# B&R Automation Studio project x20ost (part 8)

#### bnrtcpserver.c
```c
/********************************************************************
 * COPYRIGHT -- Kontora
 ********************************************************************
 * Program: bnrmain
 * File: bnrlsens.c
 * Author: Abramenya
 * Created: January 19, 2009
 *******************************************************************/

#include "bnrtcpserver.h"
#ifdef _DEFAULT_INCLUDES
 #include <AsDefault.h>
#endif
#ifdef WIN32
DWORD dwThreadId;
//void TcpOpen(TcpOpen_typ *pServer){pServer->status=0;}
SOCKET sClient;
DWORD WINAPI GetArm(PVOID pVoid);
void TcpClose(TcpClose_typ *pCL){};
void TcpServer(TcpServer_typ *pServer){pServer->identclnt=pServer->ident;pServer->status=0;}
void TcpOpen(TcpOpen_typ *pServer)
{
	BOOL    bInterface = FALSE;
    WSADATA wsd;
	int iAddrSize;
	struct sockaddr_in local,client;
	struct sockaddr_in server;
    struct hostent *host = NULL;
	pServer->status = 1;
	if (WSAStartup(MAKEWORD(2,2), &wsd) != 0)
    {
        printf("Failed to load Winsock!\n");
        return ;
    }
	pServer->sListen = socket(AF_INET, SOCK_STREAM, IPPROTO_TCP);
    if (pServer->sListen == SOCKET_ERROR)
    {
        printf("socket() failed: %d\n", WSAGetLastError());
        return ;
    }
    if (bInterface)
    {
        //local.sin_addr.s_addr = inet_addr(pServer->pIfAddr);
		local.sin_addr.s_addr = inet_addr("0.0.0.0");
        if (local.sin_addr.s_addr == INADDR_NONE)
		{
			printf("socket() failed: %s\n", pServer->pIfAddr);
			return;
		}
    }
    else
		local.sin_addr.s_addr = htonl(INADDR_ANY);
	local.sin_family = AF_INET;
	local.sin_port = htons((u_short)pServer->port);
    if (bind(pServer->sListen, (struct sockaddr *)&local,sizeof(local)) == SOCKET_ERROR)
    {
        printf("bind() failed: %d\n", WSAGetLastError());
        return ;
    }
    listen(pServer->sListen, 8);
    iAddrSize = sizeof(client);
    //pServer->sClient = accept(pServer->sListen, (struct sockaddr *)&client,&iAddrSize);
	pServer->sClient = accept(pServer->sListen, (struct sockaddr *)&client,&iAddrSize);
    if (pServer->sClient == INVALID_SOCKET)
    {
		printf("accept() failed: %d\n", WSAGetLastError());
		return ;
    }
	sClient = pServer->sClient;
	pServer->ident = &pServer->sClient;
	Info("\n(__)CTCPS::>Connect");
	pServer->status = 0;
}
//void TcpSend(TcpSend_typ *pCL){};
void TcpSend(TcpSend_typ *pSend)
{
	int ret;
	ret = send(sClient, (char*)pSend->pData, pSend->datalen, 0);
	//Info("\n(__)ARM_0:%M",pSend->buffer);
	if (ret == 0)
	{
		//printf("Send Not Poss \n");
		//Sleep(500);
		pSend->status = 1;
		return;
	}
	else if (ret == SOCKET_ERROR)
	{
		//printf("send() failed: %d\n",WSAGetLastError());
		//Sleep(500);
		pSend->status = 1;
		return;
	}
	//Sleep(50);
	pSend->status = 0;

}
void TcpRecv(TcpRecv_typ *pRecv)
{
	int ret;
	//printf("RCV\n");
	ret = recv(sClient,(char*)pRecv->pData,pRecv->datamax , 0);
	if (ret == 0)
	{
		//Sleep(500);
		printf("recv() failed 0: %d\n", WSAGetLastError());
		pRecv->status = 1;
		return;
	}
	else if (ret == SOCKET_ERROR)
	{
		printf("recv() failed: %d\n", WSAGetLastError());
        //Sleep(500);
		pRecv->status = 1;
		return;
	}
	//printf("Reccive OK! \n");
	pRecv->recvlen = ret;
	pRecv->status = 0;
}
#endif

//_GLOBAL INT iCreate1;
_GLOBAL UINT iCreateTcp1;
void CTcpServer_Init(This,SARMINTERFACE *pArm)
{
    DECLARE_MULTI_OPEN(CTcpServer,CCyclicSystem)
	FDEFINE(DEV_TCPRM_BOX_ID,1024);
	FDEFINE(DEV_TCPBF_BOX_ID,1024);
	pB->SetBoxID(pB,DEV_TCPRM_BOX_ID);
	InitObject(CMTimer,&pT->m_nConnTMR);
	pT->m_nConnTMR.SetTimer(&pT->m_nConnTMR,DIR_TCPTOTCP,DIR_TCPTOTCP,EV_TMR_SRR_REQ,0,0,DEV_TCPRM_BOX_ID);
	pT->m_pArm = pArm;
	pT->m_dwAPortNumber = pArm->dwpPortNumber[0];
	pT->m_dwBPortNumber = pArm->dwpPortNumber[1];
	strcpy(pT->m_stTcpAddr,pArm->chTcpAddr);
	#ifdef DEB_CTcpServer
	Info("\n\r(__)CTcpS::>Create Tcp.PA: %d.PB: %d. Addr[%s]",&pT->m_dwAPortNumber,&pT->m_dwBPortNumber,pT->m_stTcpAddr);
    #endif
	memset(&pT->m_npListen,0,sizeof(TcpOpen_typ));
	memset(&pT->m_npServer,0,sizeof(TcpServer_typ));
	memset(&pT->m_npSend,0,sizeof(TcpSend_typ));
	pT->m_npListen.enable  = TRUE;
	pT->m_npListen.port    = pT->m_dwAPortNumber;
	pT->m_npListen.pIfAddr = 0;
	pT->m_npListen.status  = 1;
	pT->m_npListen.options = 0;

	pT->m_blSState = TRUE;
	pT->m_blRState = TRUE;
	pT->m_bSrvState = DRV_ST_DISC;

	pT->m_nConnTMR.OnTimer(&pT->m_nConnTMR,100);
    #ifdef WIN32
	CreateThread(NULL,0,GetArm ,pT,0,&dwThreadId);
	#endif
}
_GLOBAL TcpServer_typ sServer;
_GLOBAL TcpRecv_typ sRecc;
BOOL CTcpServer_Open(This)
{
	DECLARE_MULTI_OPEN(CTcpServer,CCyclicSystem)

	if(pT->m_bSrvState==DRV_ST_DISC)
	{
	 if (pT->m_byConnReq++%2==0)
	 {
	  pT->CloseRecc(pT);
	  pT->CloseSend(pT);
	  pT->CloseOpen(pT);
	 }
	 pT->Listen(pT);
	}

	if(pT->m_bSrvState==DRV_ST_OPEN)
	{
	 pT->m_npServer.enable  = 1;
	 pT->m_npServer.ident   = pT->m_npListen.ident;
	 pT->m_npServer.backlog = 1;
	 pT->m_npServer.pIpAddr = pT->m_stTcpAddr;
     TcpServer(&pT->m_npServer);
	 memcpy(&sServer,&pT->m_npServer,sizeof(TcpServer_typ));
     if(pT->m_npServer.status==0)
	 {

	  //if(pT->m_bSrvState==DRV_ST_OPEN)
      pT->m_npRecc.enable   = 1;
      pT->m_npRecc.ident    = pT->m_npServer.identclnt;
	  pT->m_npRecc.datamax  = sizeof(SMESSAGE)-10;
	  pT->m_npRecc.flags     = 0;

	  pT->m_npSend.enable   = 1;
	  pT->m_npSend.ident    = pT->m_npServer.identclnt;
	  pT->m_npSend.datalen  = sizeof(SMESSAGE);
	  pT->m_npSend.flags    = 0;
	  pT->m_bSrvState = DRV_ST_CONN;
	  pT->m_blSState = TRUE;
	  //pT->Connect(pT);
	  pT->SendSMessage(pT,DEV_KPMDL_BOX_ID,DIR_PHTOKP,PH_CALL_REQ);
  	  return TRUE;
	 }
	}
    return TRUE;
}
_GLOBAL TcpOpen_typ sOpen;
_GLOBAL INT iListen;
BOOL CTcpServer_Listen(This)
{
    DECLARE_MULTI_OPEN(CTcpServer,CCyclicSystem)
	iListen++;
	pT->m_npListen.enable  = TRUE;
	pT->m_npListen.port    = pT->m_dwAPortNumber;
	pT->m_npListen.pIfAddr = 0;
	pT->m_npListen.status  = 1;
	pT->m_npListen.options = 0;
    TcpOpen(&pT->m_npListen);
 	memcpy(&sOpen,&pT->m_npListen,sizeof(TcpOpen_typ));
	if(pT->m_npListen.status==32602){pT->Close(pT,pT->m_npListen.ident);};
	if(pT->m_npListen.status==0)
	{
	 pT->m_bSrvState = DRV_ST_OPEN;
	 return TRUE;
	}
}

_GLOBAL TcpSend_typ sSend;
_GLOBAL INT iCTcpSrvVal,iCTcpSendCh;
//_GLOBAL INT iLnSSend;
BOOL CTcpServer_SendMessage(This,SMESSAGE *pMsg)
{
    DECLARE_MULTI_OPEN(CTcpServer,CCyclicSystem)
	iCTcpSrvVal++;
	//pT->m_blSState = TRUE;
	//pT->AddCRC(pT,TRUE,pMsg);
	pT->m_npSend.pData   = &pMsg->m_sbyInfo[0];
	pT->m_npSend.datalen = pMsg->m_swLen-9;
	TcpSend(&pT->m_npSend);
	memcpy(&sSend,&pT->m_npSend,sizeof(TcpSend_typ));
	if(pT->m_npSend.status!=0)
	{
	 if(pT->m_npSend.status==32609)
	 {
		 iCTcpSendCh++;
		 pT->CloseSend(pT);
		 pT->CloseRecc(pT);
		 pT->CloseOpen(pT);
		 pT->Disconnect(pT);
	 }
	 pT->m_blSState = FALSE;
	 return FALSE;
    }
	return TRUE;
}
_GLOBAL INT iPSend;
//_GLOBAL INT iLnPSend;
void CTcpServer_PostSend(This)
{
    DECLARE_MULTI_OPEN(CTcpServer,CCyclicSystem)
	iPSend++;
	TcpSend(&pT->m_npSend);
	memcpy(&sSend,&pT->m_npSend,sizeof(TcpSend_typ));
  	if(pT->m_npSend.status==0)pT->m_blSState = TRUE;
	if(pT->m_npSend.status==32609){iCTcpSendCh++;pT->CloseSend(pT);pT->CloseRecc(pT);pT->CloseOpen(pT);pT->Disconnect(pT);}
}

//_GLOBAL INT iCTcpCliVal;
_GLOBAL INT iCTcpInData;
//_GLOBAL SMESSAGE sMS;

BOOL CTcpServer_GetMessage(This,SMESSAGE *pMsg)
{
    DECLARE_MULTI_OPEN(CTcpServer,CCyclicSystem)
	pT->m_npRecc.pData = &pMsg->m_sbyInfo[0];
	TcpRecv(&pT->m_npRecc);
	memcpy(&sRecc,&pT->m_npRecc,sizeof(TcpRecv_typ));
	if(pT->m_npRecc.status==0)
	{
	 iCTcpInData++;
	 pMsg->m_swLen  = 9 + pT->m_npRecc.recvlen;
	 pMsg->m_sbyFor = DIR_PHTO101;
	 if (pMsg->m_swLen<300) return TRUE; else return FALSE;
	}
	else
    return FALSE;
}
_GLOBAL INT nReceiveThreadTcp,nSendThreadTcp,nSNDUR;
void CTcpServer_SendThread(This)
{
    DECLARE_MULTI_OPEN(CTcpServer,CCyclicSystem)
	nSendThreadTcp++;
	if(pT->m_bSrvState==DRV_ST_CONN)
    {
	 if(pT->m_blSState==FALSE)
	 	 pT->PostSend(pT);else
	 if(FGET(DEV_TCPBF_BOX_ID,&pT->m_sMsg0))
	 {
	  //Info("\n(__)CTcpR::>TX:%M",&pT->m_sMsg);
	  nSNDUR++;
	  pT->AddCRC(pT,TRUE,&pT->m_sMsg0);
      pT->SendMessage(pT,&pT->m_sMsg0);
	 }
	}
}
_GLOBAL INT nCheckOpenTcp,nCheckSendCheck;
void CTcpServer_ReceiveThread(This)
{
    DECLARE_MULTI_OPEN(CTcpServer,CCyclicSystem)
	nReceiveThreadTcp++;
	if(pT->m_bSrvState==DRV_ST_CONN)
	if(pT->GetMessage(pT,&pT->m_sMsg)==TRUE)
	{
	  nCheckOpenTcp = 0;
	  pT->m_nConnTMR.OnTimer(&pT->m_nConnTMR,100);
	  //Info("\n(__)CTCPM::>RX:%M",&pT->m_sMsg);
	  if(pT->CheckCRC(pT,FALSE,&pT->m_sMsg)==TRUE)
	  {
	   pT->m_sMsg.m_swLen -= 4;
	   pT->m_sMsg.m_sbyFrom       = DIR_PHMDL;
	   pT->m_sMsg.m_sbyFor        = DIR_PHTOMS;
	   pT->m_sMsg.m_sbyIntType    = 0;
	   pT->m_sMsg.m_sbyServerID   = 0;
	   pT->m_sMsg.m_sbyType       = PH_SCMD_REQ;
	   pT->m_sMsg.m_sbyDirection  = 0;
	   pT->m_sMsg.m_sbySensor     = 0;
       FPUT(DEV_MSMDL_BOX_ID,(BYTE*)&pT->m_sMsg);
	  }
	}
}
//_GLOBAL INT iPRecv;
BOOL CTcpServer_PostGet(This)
{
    DECLARE_MULTI_OPEN(CTcpServer,CCyclicSystem)
	return FALSE;
}
//_GLOBAL Tcpclose_typ sClose;
BOOL CTcpServer_Close(This,UDINT uModule)
{
    DECLARE_MULTI_OPEN(CTcpServer,CCyclicSystem)
    BOOL res = TRUE;
	pT->m_bSrvState      = DRV_ST_DISC;
	pT->m_npClose.enable = TRUE;
	pT->m_npClose.ident  = uModule;
	pT->m_npClose.how    = 3;
	TcpClose(&pT->m_npClose);
	//pT->Init(pT,pT->m_pArm);
	//memcpy(&sClose,&pT->m_npClose,sizeof(Tcpclose_typ));
	if(pT->m_npClose.status==0)return TRUE;
    return FALSE;
}
BOOL CTcpServer_CloseOpen(This)
{
    DECLARE_MULTI_OPEN(CTcpServer,CCyclicSystem)
	BOOL res =pT->Close(pT,pT->m_npListen.ident);
	pT->m_bSrvState = DRV_ST_DISC;
	memset(&pT->m_npSend,0,sizeof(TcpSend_typ));
	return res;
}
BOOL CTcpServer_CloseSend(This)
{
    DECLARE_MULTI_OPEN(CTcpServer,CCyclicSystem)
	BOOL res =pT->Close(pT,pT->m_npSend.ident);
	pT->m_bSrvState = DRV_ST_DISC;
	memset(&pT->m_npSend,0,sizeof(TcpSend_typ));
	memset(&sSend,0,sizeof(TcpRecv_typ));
	return res;
}
BOOL CTcpServer_CloseRecc(This)
{
    DECLARE_MULTI_OPEN(CTcpServer,CCyclicSystem)
	BOOL res = pT->Close(pT,pT->m_npRecc.ident);
	pT->m_bSrvState = DRV_ST_DISC;
	memset(&pT->m_npRecc,0,sizeof(TcpRecv_typ));
	memset(&sRecc,0,sizeof(TcpRecv_typ));
    return res;
}
BOOL CTcpServer_CheckSend(This)
{
    DECLARE_MULTI_OPEN(CTcpServer,CCyclicSystem)
    return TRUE;
}
void CTcpServer_WordXCHG(This,SMESSAGE *pMsg)
{
	DECLARE_MULTI_OPEN(CTcpServer,CCyclicSystem)
    #ifndef WIN32
	BYTE byTmp,*pW = (BYTE*)pMsg;
	byTmp = pW[0];
	pW[0] = pW[1];
	pW[1] = byTmp;
    #endif
}
BOOL CTcpServer_CheckCRC(This,BOOL blCrc,SMESSAGE *pMsg)
{
	DECLARE_MULTI_OPEN(CTcpServer,CCyclicSystem)
	DWORD dwCrc = 0;
	WORD wLen = pMsg->m_swLen;
	BYTE *pR = (BYTE*)&dwCrc;
	BYTE *pM = (BYTE*)pMsg;
	BYTE *pCRC = &pM[wLen-4];
    #ifndef WIN32
	pR[3] = pCRC[0];
	pR[2] = pCRC[1];
	pR[1] = pCRC[2];
	pR[0] = pCRC[3];
    #else
	memcpy(&dwCrc,pCRC,4);
    #endif
	if(dwCrc==pT->ClcCRC(pT,blCrc,pMsg)) return TRUE;
	return FALSE;
}
DWORD CTcpServer_ClcCRC(This,BOOL blCrc,SMESSAGE *pMsg)
{
    DECLARE_MULTI_OPEN(CTcpServer,CCyclicSystem)
	WORD i;
	WORD wLen;
	DWORD dwCrc = 0;
	//BYTE *pCRC,*pM = (BYTE*)&pMsg;
	BYTE *pCRC,*pM = (BYTE*)&pMsg->m_sbyInfo[0];
	if (blCrc) pMsg->m_swLen += 4;
	//wLen = pMsg->m_swLen-4;
	wLen = pMsg->m_swLen-4-9;
	pCRC = &pM[wLen];
	for(i=0;i<wLen;i++)
	{
	 dwCrc += pM[i];
	 if(i>700)
		 break;
	}
	return dwCrc;
}
void CTcpServer_AddCRC(This,BOOL blCrc,SMESSAGE *pMsg)
{
	DECLARE_MULTI_OPEN(CTcpServer,CCyclicSystem)
	DWORD dwCrc = 0;
	WORD wLen = pMsg->m_swLen;
	BYTE *pR = (BYTE*)&dwCrc;
	BYTE *pM = (BYTE*)pMsg;
	BYTE *pCRC = &pM[wLen];
	dwCrc = pT->ClcCRC(pT,blCrc,pMsg);
    #ifndef WIN32
	pCRC[3] = pR[0];
	pCRC[2] = pR[1];
	pCRC[1] = pR[2];
	pCRC[0] = pR[3];
    #else
	memcpy(pCRC,pR,4);
    #endif
}

BOOL CTcpServer_EventHandler(This,SMESSAGE *pMsg)
{
    DECLARE_MULTI_OPEN(CTcpServer,CCyclicSystem)
	//SHORTMESSAGE m_sMsg;
	switch(pMsg->m_sbyFor)
	{
      case DIR_MSTOTCP:
	       #ifdef DEB_CTcpServer
		   Info("\n(__)CTCPR::>OUTP::%M",pMsg);
		   #endif
		   FPUT(DEV_TCPBF_BOX_ID,pMsg);
	  break;
	  case DIR_TCPTOTCP:
	       if (pMsg->m_sbyType==EV_TMR_SRR_REQ)
		   {

 		    pT->Open(pT);
			pT->m_nConnTMR.OnTimer(&pT->m_nConnTMR,100);
			//if (nCheckOpenTcp%4==0)
			{
             nCheckSendCheck++;
			 pT->m_sMsg0.m_swLen      = 9+3;
			 pT->m_sMsg0.m_sbyInfo[0] = 0x55;
			 pT->m_sMsg0.m_sbyInfo[1] = 0xaa;
			 pT->m_sMsg0.m_sbyInfo[2] = 0x55;
			 pT->m_sMsg0.m_sbyInfo[3] = 3;
			 pT->m_sMsg0.m_sbyInfo[4] = 4;
			 ////SendMessage()
			 FPUT(DEV_TCPBF_BOX_ID,&pT->m_sMsg0);
			}
			nCheckOpenTcp++;
		   }
	  break;
	  default:
	  break;
	}
	return TRUE;
}
void CTcpServer_CyclicProc(This)
{
    DECLARE_MULTI_OPEN(CTcpServer,CCyclicSystem)
    #ifndef WIN32
	pT->SendThread(pT);
	pT->ReceiveThread(pT);
    #else
	pT->SendThread(pT);
    #endif
}
void CTcpServer_SendSMessage(This,BYTE byBox,BYTE byFor,BYTE byType)
{
    DECLARE_MULTI_OPEN(CTcpServer,CCyclicSystem)
	SHORTMESSAGE m_sMsg;
	m_sMsg.m_swLen        = 9;
	m_sMsg.m_sbyFrom      = DIR_PHMDL;
	m_sMsg.m_sbyFor       = byFor;
	m_sMsg.m_sbyIntType   = 0;
	m_sMsg.m_sbyServerID  = 0;
	m_sMsg.m_sbyType      = byType;
	m_sMsg.m_sbyDirection = 0;
	m_sMsg.m_sbySensor    = 0;
	FPUT(byBox,(BYTE*)&m_sMsg);
    #ifdef DEB_CTcpServer
	Info("\n(__)CTCPR::>OUTT::%M",&m_sMsg);
    #endif
}
void CTcpServer_Connect(This)
{
    DECLARE_MULTI_OPEN(CTcpServer,CCyclicSystem)
    SHORTMESSAGE m_sMsg;
	m_sMsg.m_swLen        = 9;
	m_sMsg.m_sbyFrom      = DIR_PHMDL;
	m_sMsg.m_sbyFor       = DIR_PHTO101P;
	m_sMsg.m_sbyIntType   = 0;
	m_sMsg.m_sbyServerID  = 0;
	m_sMsg.m_sbyType      = PH_CONN_IND;
	m_sMsg.m_sbyDirection = 0;
	m_sMsg.m_sbySensor    = 0;
	FPUT(DEV_101MD_BOX_ID,(BYTE*)&m_sMsg);
    #ifdef DEB_CTcpServer
	Info("\n(__)CTCPR::>OUTT::%M",&m_sMsg);
    #endif
}
void CTcpServer_Disconnect(This)
{
    DECLARE_MULTI_OPEN(CTcpServer,CCyclicSystem)
    SHORTMESSAGE m_sMsg;
	m_sMsg.m_swLen        = 9;
	m_sMsg.m_sbyFrom      = DIR_PHMDL;
	m_sMsg.m_sbyFor       = DIR_PHTO101P;
	m_sMsg.m_sbyIntType   = 0;
	m_sMsg.m_sbyServerID  = 0;
	m_sMsg.m_sbyType      = PH_DISC_IND;
	m_sMsg.m_sbyDirection = 0;
	m_sMsg.m_sbySensor    = 0;
	FPUT(DEV_101MD_BOX_ID,(BYTE*)&m_sMsg);
    #ifdef DEB_CTcpServer
	Info("\n(__)CTCPR::>OUTT::%M",&m_sMsg);
    #endif
}
void CTcpServer_CTcpServer(This)
{
    DECLARE_MULTI_OPEN(CTcpServer,CCyclicSystem)
	DECLARE_REGISTRATION(CTcpServer,Init)
	DECLARE_REGISTRATION(CTcpServer,PostSend)
	DECLARE_REGISTRATION(CTcpServer,PostGet)
	DECLARE_REGISTRATION(CTcpServer,SendMessage)
	DECLARE_REGISTRATION(CTcpServer,GetMessage)
	DECLARE_REGISTRATION(CTcpServer,CheckSend)
	DECLARE_REGISTRATION(CTcpServer,Open)
	DECLARE_REGISTRATION(CTcpServer,Listen)
	DECLARE_REGISTRATION(CTcpServer,Close)
	DECLARE_REGISTRATION(CTcpServer,CloseSend)
	DECLARE_REGISTRATION(CTcpServer,CloseRecc)
	DECLARE_REGISTRATION(CTcpServer,WordXCHG)
	DECLARE_REGISTRATION(CTcpServer,AddCRC)
	DECLARE_REGISTRATION(CTcpServer,CheckCRC)
	DECLARE_REGISTRATION(CTcpServer,ClcCRC)
	DECLARE_REGISTRATION(CTcpServer,ReceiveThread)
	DECLARE_REGISTRATION(CTcpServer,SendThread)
	DECLARE_REGISTRATION(CTcpServer,CloseOpen)
	DECLARE_REGISTRATION(CTcpServer,Connect)
	DECLARE_REGISTRATION(CTcpServer,Disconnect)
	DECLARE_REGISTRATION(CTcpServer,SendSMessage)
	DECLARE_VIRTUAL_FUNC(CTcpServer,EventHandler)
	DECLARE_VIRTUAL_FUNC(CTcpServer,CyclicProc)
}
void CTcpServer_DCTcpServer(This)
{
	DECLARE_MULTI_OPEN(CTcpServer,CCyclicSystem)
}
DECLARE_MULTI_CREATE(CTcpServer,CCyclicSystem)
#ifdef WIN32
DWORD WINAPI GetArm(PVOID pVoid)
{
	CTcpServer *pT = (CTcpServer*)pVoid;
	while(1)
	{
	 pT->ReceiveThread(pT);
	 //pT->SendThread(pT);
	 //Sleep(50);
     //printf("\nGetArm");
	}
	return 0;
}
#endif
```

#### bnrtu.h
```c
/********************************************************************
 * COPYRIGHT -- Kontora
 ********************************************************************
 * Program: bnrmain
 * File: bnraninput.h
 * Author: Abramenya
 * Created: January 19, 2009
 *******************************************************************/

#ifndef __TU_H__
#define __TU_H__
#include "typedefs.h"
#include "bnrdevice.h"
#include "bnrpin.h"
#include "bnrdevtu.h"
Class CTu
{
	 void (*CCTu)(This);
	 void (*DCTu)(This);
Public
	 Virtual BOOL (*EventHandler)(This,SMESSAGE *pMsg);
	 Virtual void (*InitTCHN)(This,PVOID psTable);
     Virtual void (*PreProc)(This);
	 Virtual void (*Processing)(This);
     Virtual void (*PostProc)(This);
	 Virtual PVOID (*GetData)(This,BYTE *pData,WORD *nLen);
Public
     STUMPARAM *pP;
     CDevTU *pTU0;
	 DECLARE_IMPLEMENT_BASE(CDevice)
}
DECLARE_DEFINITION(CTu)
#endif
```

#### bnrtemper.c
```c
/********************************************************************
 * COPYRIGHT -- Kontora
 ********************************************************************
 * Program: bnrmain
 * File: bnrlsens.c
 * Author: Abramenya
 * Created: January 19, 2009
 *******************************************************************/

#include "bnrtemper.h"
#include "bnrmain.h"
#ifdef _DEFAULT_INCLUDES
 #include <AsDefault.h>
#endif
_GLOBAL BYTE nFSignal;
void CTemper_InitTCHN(This,PVOID psTable)
{
    DECLARE_MULTI_OPEN(CTemper,CDevice)
	CSlot *pSL;
	CPin *m_pPN0;
	BOOL *m_pbVL0;
	CComputer *pCM = pB->m_pComputer;

    pT->pP = (STTMPARAM*)psTable;
	pB->m_nSize = 2*sizeof(WORD);

	pSL          = pCM->GetSlot(pCM,pT->pP->bySlot);
	m_pPN0       = pSL->GetPin(pSL->pChld,pT->pP->byPin);
    pT->m_pwVL0 = (WORD*)m_pPN0->GetAddrPin(m_pPN0->pChld);

    #ifdef DEB_CTemper
	//Info("\n(%b)CTLSG::>Create TeleSignal.",&pB->m_byID);
    #endif
}
void CTemper_PreProc(This)
{
    DECLARE_MULTI_OPEN(CTemper,CDevice)
	pT->pP->sDT.wParam = *pT->m_pwVL0;
}
_GLOBAL INT nTSCH;
void CTemper_Processing(This)
{
	DECLARE_MULTI_OPEN(CTemper,CDevice)
}
void CTemper_PostProc(This)
{
	DECLARE_MULTI_OPEN(CTemper,CDevice)
	BOOL res = FALSE;
}
BYTE CTemper_CheckTS(This)
{
    DECLARE_MULTI_OPEN(CTemper,CDevice)
    //return pB->m_pPN->GetState(pB->m_pPN);
	return 0;
}
BOOL CTemper_EventHandler(This,SMESSAGE *pMsg)
{
    DECLARE_MULTI_OPEN(CTemper,CDevice)
    BYTE byID = pMsg->m_sbySensor;
	BYTE byParamType = pMsg->m_sbyInfo[3];
    #ifdef DEB_CTemper
	Info("\n(%b)CTLSG::>INPT::%M",&pB->m_byID,pMsg);
    #endif
	switch(pMsg->m_sbyFor)
	{
	  case DIR_101TOKP:
		   switch(pMsg->m_sbyType)
		   {
		    case PL_DATA_IND:
				 //Info("\n(%b)CTLSG::>DL_DATA_IND::>%M",&pB->m_byID,pMsg);
				 switch(byParamType)
				 {
				   case EN_SET_PERIOD:
					    //pT->m_byCSetPulce = pMsg->m_sbyInfo[3];
					    //pT->m_bySetPulce  = pT->m_byCSetPulce;
				   break;
				   case EN_REM_PERIOD:
					    //pT->m_byRemPulce  = pMsg->m_sbyInfo[3];
						//pT->m_byCRemPulce = pT->m_byRemPulce;
				   break;
				   case EN_PIN_ALMODE:
                        //pT->m_byAlarmMode = pMsg->m_sbyInfo[3];
				   break;
				   default:
				   break;
				 }
		    break;
			default:
            break;
		   }
      break;
	  case DIR_101MD:
	  break;
	  default:
	  break;
	}
	return TRUE;
}
void CTemper_SetInPinEvent(This)
{
    DECLARE_MULTI_OPEN(CTemper,CDevice)
}
void CTemper_SaveAlarmPin(This)
{
	DECLARE_MULTI_OPEN(CTemper,CDevice)
}
void CTemper_SendObsrveMsg(This)
{
    DECLARE_MULTI_OPEN(CTemper,CDevice)
}
/*
typedef struct _tagTTMData
{
UINT wJob;
UINT wParam;
}STTMDATA;
*/
PVOID CTemper_GetData(This,BYTE *pData,WORD *nLen)
{
    DECLARE_MULTI_OPEN(CTemper,CDevice)
	pB->GetWordParam(pB,(BYTE*)&pT->pP->sDT.wJob,&pData[0]);
	pB->GetWordParam(pB,(BYTE*)&pT->pP->sDT.wParam,&pData[2]);
	*nLen += pB->m_nSize;if (*nLen>350) *nLen=0;
	return pData;
}
void CTemper_CTemper(This)
{
    DECLARE_MULTI_OPEN(CTemper,CDevice)
	DECLARE_REGISTRATION(CTemper,CheckTS)
	DECLARE_VIRTUAL_FUNC(CTemper,EventHandler)
	DECLARE_VIRTUAL_FUNC(CTemper,InitTCHN)
	DECLARE_VIRTUAL_FUNC(CTemper,PreProc)
	DECLARE_VIRTUAL_FUNC(CTemper,Processing)
	DECLARE_VIRTUAL_FUNC(CTemper,PostProc)
	DECLARE_VIRTUAL_FUNC(CTemper,SetInPinEvent)
	DECLARE_VIRTUAL_FUNC(CTemper,SaveAlarmPin)
	DECLARE_VIRTUAL_FUNC(CTemper,SendObsrveMsg)
	DECLARE_VIRTUAL_FUNC(CTemper,GetData)
}
void CTemper_DCTemper(This)
{
	DECLARE_MULTI_OPEN(CTemper,CDevice)
}
DECLARE_MULTI_CREATE(CTemper,CDevice)
```

#### bnrtemper.h
```c
/********************************************************************
 * COPYRIGHT -- Kontora
 ********************************************************************
 * Program: bnrmain
 * File: bnraninput.h
 * Author: Abramenya
 * Created: January 19, 2009
 *******************************************************************/

#ifndef __TEMPER_H__
#define __TEMPER_H__
#include "typedefs.h"
#include "bnrdevice.h"
#include "bnrpin.h"

Class CTemper
{
	 void (*CCTemper)(This);
	 void (*DCTemper)(This);
Public
     BYTE (*CheckTS)(This);
	 Virtual BOOL (*EventHandler)(This,SMESSAGE *pMsg);
	 Virtual void (*InitTCHN)(This,PVOID psTable);
     Virtual void (*PreProc)(This);
	 Virtual void (*Processing)(This);
     Virtual void (*PostProc)(This);
	 Virtual void (*SetInPinEvent)(This);
	 Virtual void (*SaveAlarmPin)(This);
	 Virtual void (*SendObsrveMsg)(This);
	 Virtual PVOID (*GetData)(This,BYTE *pData,WORD *nLen);
Public
     STTMPARAM *pP;
	 WORD *m_pwVL0;
	 DECLARE_IMPLEMENT_BASE(CDevice)
}
DECLARE_DEFINITION(CTemper)
#endif
```

#### bnrts.c
```c
/********************************************************************
 * COPYRIGHT -- Kontora
 ********************************************************************
 * Program: bnrmain
 * File: bnrlsens.c
 * Author: Abramenya
 * Created: January 19, 2009
 *******************************************************************/

#include "bnrts.h"
#include "bnrmain.h"
#ifdef _DEFAULT_INCLUDES
 #include <AsDefault.h>
#endif
_GLOBAL BYTE nFSignal;
void CTs_InitTCHN(This,PVOID psTable)
{
    DECLARE_MULTI_OPEN(CTs,CDevice)
	CSlot *pSL;
	CPin *m_pPN0;
	BOOL *m_pbAVL0;
	CComputer *pCM = pB->m_pComputer;
	pT->pP = (STSMPARAM*)psTable;
	pB->m_nSize = 1;
    //Вход
	pSL          = pCM->GetSlot(pCM,pT->pP->bySlot);
	m_pPN0       = pSL->GetPin(pSL->pChld,pT->pP->byPin);
    m_pbAVL0 = (BOOL*)m_pPN0->GetAddrPin(m_pPN0->pChld);
	New(sizeof(CDevTS),pT->pTS0);
	InitObject(CDevTS,pT->pTS0);
    pT->pTS0->Init(pT->pTS0,m_pPN0, m_pbAVL0,pT->pP->byID,0,EN_OPEN,PRI_HI,pT->pP->byCRemPulce,pT->pP->byCSetPulce,EN_AL_TO_AL);
	pT->pTS0->SetTS(pT->pTS0,DEV_MSMDL_BOX_ID,DIR_MSTOMS,EV_CHNG_PIN_REQ);

    #ifdef DEB_CTs
	//Info("\n(%b)CTLSG::>Create TeleSignal.",&pB->m_byID);
    #endif
}
void CTs_PreProc(This)
{
    DECLARE_MULTI_OPEN(CTs,CDevice)
	pT->pTS0->Run(pT->pTS0);
}
_GLOBAL INT nTSCH;
void CTs_Processing(This)
{
	DECLARE_MULTI_OPEN(CTs,CDevice)
}
void CTs_PostProc(This)
{
	DECLARE_MULTI_OPEN(CTs,CDevice)
	BOOL res = FALSE;
}
BYTE CTs_CheckTS(This)
{
    DECLARE_MULTI_OPEN(CTs,CDevice)
	//return pB->m_pPN->GetState(pB->m_pPN);
	return 0;
}
BOOL CTs_EventHandler(This,SMESSAGE *pMsg)
{
    DECLARE_MULTI_OPEN(CTs,CDevice)
	SKPEVENT pEV;
    #ifdef DEB_CTs
	//Info("\n(%b)CTLSG::>INPT::%M",&pB->m_nCD.wDeviceID,pMsg);
    #endif
	switch(pMsg->m_sbyFor)
	{
	  case DIR_MSTODV:
		   switch(pMsg->m_sbyType)
		   {
		    case PL_DATA_IND:
				 switch(pB->m_nCD.byParam0)
				 {
                   case CTR_TR:
				   break;
				   case CTR_TU:
					    //if (pB->m_nCD.wParam0==1)
						//{
						// pT->pTU0->SetPin(pT->pTU0);
						//}else
					    //if (pB->m_nCD.wParam0==0)
						//{
						// pT->pTU0->InvPin(pT->pTU0);
						//}
				   break;
				   default:
				   break;
				 }
		    break;
			case EV_CHNG_PIN_REQ:
 				 memcpy(&pEV,&pMsg->m_sbyInfo[0],sizeof(SKPEVENT));
				 switch (pEV.byType)
				 {
				    case REG_SOFTU_ADDR:
						//if ((pEV.byCause==EV_0T1_ST)&&(pEV.byAddr==0))
						//	pT->pP->sDT.byParam = 1;else
						//if ((pEV.byCause==EV_1T0_ST)&&(pEV.byAddr==0))
						//	pT->pP->sDT.byParam = 0;
					break;
					case REG_SOFTS_ADDR:
						//Активность входа
						if ((pEV.byCause==EV_0T1_CH)&&(pEV.byAddr==0))
						{
						 pT->pP->sDT.byParam = 1;
						} else
						if ((pEV.byCause==EV_1T0_CH)&&(pEV.byAddr==0))
						{
						 pT->pP->sDT.byParam = 0;
						}
					break;
				 }
			break;
			default:
            break;
		   }
      break;
	  case DIR_101MD:
	  break;
	  default:
	  break;
	}
	return TRUE;
}
PVOID CTs_GetData(This,BYTE *pData,WORD *nLen)
{
    DECLARE_MULTI_OPEN(CTs,CDevice)
	pData[0] = pT->pP->sDT.byParam;
	*nLen += pB->m_nSize;if (*nLen>350) *nLen=0;
	return pData;
}
void CTs_CTs(This)
{
    DECLARE_MULTI_OPEN(CTs,CDevice)
	DECLARE_VIRTUAL_FUNC(CTs,EventHandler)
	DECLARE_VIRTUAL_FUNC(CTs,InitTCHN)
	DECLARE_VIRTUAL_FUNC(CTs,PreProc)
	DECLARE_VIRTUAL_FUNC(CTs,Processing)
	DECLARE_VIRTUAL_FUNC(CTs,PostProc)
	DECLARE_VIRTUAL_FUNC(CTs,GetData)
}
void CTs_DCTs(This)
{
	DECLARE_MULTI_OPEN(CTs,CDevice)
}
DECLARE_MULTI_CREATE(CTs,CDevice)
```

#### bnrts.h
```c
/********************************************************************
 * COPYRIGHT -- Kontora
 ********************************************************************
 * Program: bnrmain
 * File: bnraninput.h
 * Author: Abramenya
 * Created: January 19, 2009
 *******************************************************************/

#ifndef __TS_H__
#define __TS_H__
#include "typedefs.h"
#include "bnrdevice.h"
#include "bnrpin.h"
#include "bnrdevts.h"
Class CTs
{
	 void (*CCTs)(This);
	 void (*DCTs)(This);
Public
	 Virtual BOOL (*EventHandler)(This,SMESSAGE *pMsg);
	 Virtual void (*InitTCHN)(This,PVOID psTable);
     Virtual void (*PreProc)(This);
	 Virtual void (*Processing)(This);
     Virtual void (*PostProc)(This);
	 Virtual PVOID (*GetData)(This,BYTE *pData,WORD *nLen);
Public
     STSMPARAM *pP;
     CDevTS *pTS0;
	 DECLARE_IMPLEMENT_BASE(CDevice)
}
DECLARE_DEFINITION(CTs)
#endif
```

#### bnrtu.c
```c
/********************************************************************
 * COPYRIGHT -- Kontora
 ********************************************************************
 * Program: bnrmain
 * File: bnrlsens.c
 * Author: Abramenya
 * Created: January 19, 2009
 *******************************************************************/

#include "bnrtu.h"
#include "bnrmain.h"
#ifdef _DEFAULT_INCLUDES
 #include <AsDefault.h>
#endif
_GLOBAL BYTE nFSignal;
void CTu_InitTCHN(This,PVOID psTable)
{
    DECLARE_MULTI_OPEN(CTu,CDevice)
	CSlot *pSL;
	CPin *m_pPN0;
	BOOL *m_pbVL0;
	CComputer *pCM = pB->m_pComputer;
	pT->pP = (STUMPARAM*)psTable;
	pB->m_nSize = 1;

    //Выход запуска
	pSL          = pCM->GetSlot(pCM,pT->pP->bySlot);
	m_pPN0       = pSL->GetPin(pSL->pChld,pT->pP->byPin);
    m_pbVL0 = (BOOL*)m_pPN0->GetAddrPin(m_pPN0->pChld);
	New(sizeof(CDevTU),pT->pTU0);
	InitObject(CDevTU,pT->pTU0);
    pT->pTU0->Init(pT->pTU0,m_pbVL0,pT->pP->byID,0,EN_OPEN,pT->pP->byPulceType,pT->pP->byCSetPulce);
	pT->pTU0->SetTU(pT->pTU0,DEV_MSMDL_BOX_ID,DIR_MSTOMS,EV_CHNG_PIN_REQ);
    #ifdef DEB_CTu
	//Info("\n(%b)CTLSG::>Create TeleSignal.",&pB->m_byID);
    #endif
}
void CTu_PreProc(This)
{
    DECLARE_MULTI_OPEN(CTu,CDevice)
    pT->pTU0->Run(pT->pTU0);
}
_GLOBAL INT nTSCH;
void CTu_Processing(This)
{
	DECLARE_MULTI_OPEN(CTu,CDevice)
}
void CTu_PostProc(This)
{
	DECLARE_MULTI_OPEN(CTu,CDevice)
	BOOL res = FALSE;
}
BOOL CTu_EventHandler(This,SMESSAGE *pMsg)
{
    DECLARE_MULTI_OPEN(CTu,CDevice)
	SKPEVENT pEV;
    #ifdef DEB_CTu
	//Info("\n(%b)CTLSG::>INPT::%M",&pB->m_nCD.wDeviceID,pMsg);
    #endif
	switch(pMsg->m_sbyFor)
	{
	  case DIR_MSTODV:
		   switch(pMsg->m_sbyType)
		   {
		    case PL_DATA_IND:
				 switch(pB->m_nCD.byParam0)
				 {
                   case CTR_TR:
				   break;
				   case CTR_TU:
					    switch (pB->m_nCD.byParam1)
					    {
						  case 0:
					           if (pB->m_nCD.wParam0==1) pT->pTU0->SetPin(pT->pTU0); else
					           if (pB->m_nCD.wParam0==0) pT->pTU0->InvPin(pT->pTU0);
						  break;
						  case 1:
							   pT->pTU0->SetPulce(pT->pTU0);
						  break;
						  default:
						  break;
					    }
				   break;
				   default:
				   break;
				 }
		    break;
			case EV_CHNG_PIN_REQ:
 				 memcpy(&pEV,&pMsg->m_sbyInfo[0],sizeof(SKPEVENT));
				 switch (pEV.byType)
				 {
				    case REG_SOFTU_ADDR:
						if ((pEV.byCause==EV_0T1_ST)&&(pEV.byAddr==0))
							pT->pP->sDT.byParam = 1;else
						if ((pEV.byCause==EV_1T0_ST)&&(pEV.byAddr==0))
							pT->pP->sDT.byParam = 0;
					break;
					case REG_SOFTS_ADDR:
						//Активность верхнего входа
						//if ((pEV.byCause==EV_0T1_CH)&&(pEV.byAddr==0))
						//{
						// pT->pP->sDT.byParam = 1;
						//} else
						//if ((pEV.byCause==EV_1T0_CH)&&(pEV.byAddr==0))
						//{
						// pT->pP->sDT.byParam = 0;
						//}
					break;
				 }
			break;
			default:
            break;
		   }
      break;
	  case DIR_101MD:
	  break;
	  default:
	  break;
	}
	return TRUE;
}
PVOID CTu_GetData(This,BYTE *pData,WORD *nLen)
{
    DECLARE_MULTI_OPEN(CTu,CDevice)
	pData[0] = pT->pP->sDT.byParam;
	*nLen += pB->m_nSize;if (*nLen>350) *nLen=0;
	return pData;
}
void CTu_CTu(This)
{
    DECLARE_MULTI_OPEN(CTu,CDevice)
	DECLARE_VIRTUAL_FUNC(CTu,EventHandler)
	DECLARE_VIRTUAL_FUNC(CTu,InitTCHN)
	DECLARE_VIRTUAL_FUNC(CTu,PreProc)
	DECLARE_VIRTUAL_FUNC(CTu,Processing)
	DECLARE_VIRTUAL_FUNC(CTu,PostProc)
	DECLARE_VIRTUAL_FUNC(CTu,GetData)
}
void CTu_DCTu(This)
{
	DECLARE_MULTI_OPEN(CTu,CDevice)
}
DECLARE_MULTI_CREATE(CTu,CDevice)
```

#### bnrdevice.h
```c
/********************************************************************
 * COPYRIGHT -- Kontora
 ********************************************************************
 * Program: bnrmain
 * File: bnraninput.h
 * Author: Abramenya
 * Created: January 19, 2009
 *******************************************************************/

#ifndef __DEVICE_H__
#define __DEVICE_H__
#include "typedefs.h"
#include "bnrdebug.h"
#include "bnrpob.h"
#include "bnrmessage.h"
#include "bnrcomputer.h"
Class CDevice
{
	 void (*CCDevice)(This);
	 void (*DCDevice)(This);
Public
     void (*Init)(This,PVOID *psTable);
     void (*ObserveProc)(This);
	 void (*CheckAlarm)(This);
	 BOOL (*SaveChange)(This,BYTE byEvent,WORD wValue,BOOL blAlarm);
	 BOOL (*SavePinState)(This,BYTE byEvent,WORD wValue);
	 void (*SendBroadcast)(This,SKPEVENT *pEV);
	 void (*SendSMessage)(This,BYTE byBox,BYTE byFor,BYTE byType);
	 void (*Switch)(This);
	 REAL (*GetRealParam)(This,BYTE *pbyParam,BYTE *pbyOut);
	 WORD (*GetWordParam)(This,BYTE *pbyParam,BYTE *pbyOut);
	 UDINT (*GetDWordParam)(This,BYTE *pbyParam,BYTE *pbyOut);
	 BOOL (*SEventHandler)(This,SMESSAGE *pMsg);
	 BOOL (*ExtractCMD)(This,SMESSAGE *pMsg);
	 Virtual BOOL (*EventHandler)(This,SMESSAGE *pMsg);
     Virtual void (*InitTCHN)(This,PVOID psTable);
     Virtual void (*PreProc)(This);
     Virtual void (*Processing)(This);
	 Virtual void (*PostProc)(This);
	 Virtual void (*SaveAlarmPin)(This);
	 Virtual void (*SetInPinEvent)(This);
	 Virtual void (*SendObsrveMsg)(This);
	 Virtual PVOID (*GetData)(This,BYTE *pData,WORD *nLen);

	 void (*SetMsgAuto)(This,SMESSAGE*);
	 BOOL (*SetState)(This,TStateCode vNewState);
	 TStateCode (*GetStateCode)(This);
	 BOOL (*HandleEvent)(This,TEvent vEvent);
Protected
	 Virtual BOOL (*HandleTask)(This,TTask* pvTask);
	 Virtual TStateList* (*GetStateList)(This);
	 TState* (*GetState)(This);
Protected
	 BYTE v[20];
	 TState*  m_pvState;
     TStateCode m_vState;
	 TStateList *m_pStateList;
	 CMTimer m_nATmr[4];
	 DWORD m_dwTM[4];
	 BYTE  m_byAutoState;
Public
/*
{
    CDataCommand = packed record
     wDeviceID : Word;
     byParam0  : Byte;
     byParam1  : Byte;
     byParam2  : Byte;
     wParam0   : Word;
     wParam1   : Word;
     wParam2   : Word;
     fParam0   : Single;
     fParam1   : Single;
     fParam2   : Single;
    End;
}
*/
     PVOID pP;
	 BOOL m_blSetAlarm;
     BYTE m_byID;
	 BYTE m_byIID;
	 WORD m_nSize;
	 SHARDCOMPUTERTABLE *m_pPCT;
	 CDataCommand m_nCD;
     //CPin *m_pPN;
	 //PVOID m_pvValue;
	 //BOOL *m_pvAlValue;
     CComputer *m_pComputer;
	 DECLARE_IMPLEMENT
}
DECLARE_DEFINITION(CDevice)
#endif
```

#### bnrdevice.c
```c
/********************************************************************
 * COPYRIGHT -- Kontora
 ********************************************************************
 * Program: bnrmain
 * File: bnrlsens.c
 * Author: Abramenya
 * Created: January 19, 2009
 *******************************************************************/

#include "bnrdevice.h"
#include "bnrmain.h"
#ifdef _DEFAULT_INCLUDES
 #include <AsDefault.h>
#endif
//#include "bnrmain.h"
//#ifdef WIN32
char *STTS1[]  =
{
    "EV_SET_HI",
	"EV_REM_HI",
	"EV_SET_LO",
	"EV_REM_LO",
	"EV_CHG_PR",
	"EV_0T1_CH",
	"EV_1T0_CH",
	"EV_SAL_CH",
	"EV_RAL_CH",
	"EV_0T1_ST",
	"EV_1T0_ST",
	"EV_INI_CH",
	"EV_ALP_CH",
	"EV_ALS_CH",
	"EV_DSC_CH",

};
//#endif
DECLARE_TASKCHAIN(SkipDV)
{
    {EXIT_D}
};
DECLARE_STATE(BadStateDV)
{
    {EV_UNKNOWN_REQ, SkipDV}
};
DECLARE_STATELIST(StateListDV)
{
    {S_BAD, BadStateDV}
};
BOOL CDevice_SetState(This,TStateCode vNewState)
{
	 DECLARE_SINGLE_OPEN(CDevice)
     TStateList * pvList = pT->GetStateList(pC);
     pT->m_pvState = pvList[(INT16)vNewState].m_pvState;
     pT->m_vState  = vNewState;
	 //pT->v[STATE] = vNewState;
     return TRUE;
}
BOOL CDevice_HandleEvent(This,TEvent vEvent)
{
	 DECLARE_SINGLE_OPEN(CDevice)
	 TState* pvState;
     for(pvState=pT->m_pvState; pvState->m_vEvent!=EV_UNKNOWN_REQ; pvState++)
	 {
        if(pvState->m_vEvent==vEvent)
        {
            return pT->HandleTask(pC,pvState->m_pvTask);
        }
	 }
     return FALSE;
}
BOOL CDevice_HandleTask(This,TTask* pvTask)
{
	 DECLARE_SINGLE_OPEN(CDevice)
     return (*pvTask==EXIT_D)?TRUE:FALSE;
}
TStateList* CDevice_GetStateList(This)
{
	 DECLARE_SINGLE_OPEN(CDevice)
     return (TStateList*)&StateListDV;
}
TStateCode CDevice_GetStateCode(This)
{
	 DECLARE_SINGLE_OPEN(CDevice)
	 return pT->m_vState;
}
TState* CDevice_GetState(This)
{
	 DECLARE_SINGLE_OPEN(CDevice)
	 return pT->m_pvState;
}
void CDevice_SetMsgAuto(This,SMESSAGE *pMsg)
{
     DECLARE_SINGLE_OPEN(CDevice)
	 BYTE byEvent = pMsg->m_sbyType;
	 pT->HandleEvent(pT,byEvent);
}
void CDevice_SetAutoState(This,TStateCode vNewState)
{
     DECLARE_SINGLE_OPEN(CDevice)
	 pT->SetState(pT,vNewState);
}
/////////////////////////////////////////////////////////////////
BYTE byIDD;
void CDevice_Init(This,PVOID *psTable)
{
    DECLARE_SINGLE_OPEN(CDevice)
    //pT->pP       = psTable;
	//pT->m_byType = ((STKPARAM*)psTable)->byType;
	//pT->m_byID   = ((STKPARAM*)psTable)->byID;
	//pT->m_byIID  = ((STKPARAM*)psTable)->byAmParam;

	//pT->m_blSetAlarm = FALSE;
	//pT->m_byOldEvent = 0xff;
	pT->InitTCHN(pC,psTable);
}
void CDevice_Switch(This)
{
   DECLARE_SINGLE_OPEN(CDevice)
}
void CDevice_InitTCHN(This,SSWITCHTABLE *psTable){}
void CDevice_PreProc(This){}
void CDevice_Processing(This){}
void CDevice_PostProc(This){}
void CDevice_ObserveProc(This)
{
     DECLARE_SINGLE_OPEN(CDevice)
	 pT->PreProc(pC);
	 pT->Processing(pC);
	 pT->PostProc(pC);
     //if(++pT->m_byALC%20==0) pT->CheckAlarm(pT);
}
void CDevice_CheckAlarm(This)
{
     DECLARE_SINGLE_OPEN(CDevice)
}
BOOL CDevice_SEventHandler(This,SMESSAGE *pMsg)
{
	 DECLARE_SINGLE_OPEN(CDevice)
     switch(pMsg->m_sbyFor)
	 {
	  case DIR_MSTODV:
		   if (pMsg->m_sbyType==PL_DATA_IND)
		   {
            pT->ExtractCMD(pT,pMsg);
			pT->EventHandler(pC,pMsg);
		   }
	  break;
	  default:
	  break;
	 }
	 return TRUE;
}
/*
{
    CDataCommand = packed record
     wDeviceID : Word;
     byParam0  : Byte;
     byParam1  : Byte;
     byParam2  : Byte;
     wParam0   : Word;
     wParam1   : Word;
     wParam2   : Word;
     fParam0   : Single;
     fParam1   : Single;
     fParam2   : Single;
    End;
}
*/
BOOL CDevice_ExtractCMD(This,SMESSAGE *pMsg)
{
	 DECLARE_SINGLE_OPEN(CDevice)
	 CDataCommand *pCD;
	 pCD = &pT->m_nCD;
	 memset(pCD,0,11);pCD->fParam0 = pCD->fParam1 = pCD->fParam2 = 0;
 	 pT->GetWordParam(pT,&pMsg->m_sbyInfo[0],(BYTE*)&pCD->wDeviceID);
	 pCD->byParam0 = pMsg->m_sbyInfo[2];
	 pCD->byParam1 = pMsg->m_sbyInfo[3];
	 pCD->byParam2 = pMsg->m_sbyInfo[4];
	 pT->GetWordParam(pT,&pMsg->m_sbyInfo[5],(BYTE*)&pCD->wParam0);
	 pT->GetWordParam(pT,&pMsg->m_sbyInfo[7],(BYTE*)&pCD->wParam1);
	 pT->GetWordParam(pT,&pMsg->m_sbyInfo[9],(BYTE*)&pCD->wParam2);
	 pT->GetRealParam(pT,&pMsg->m_sbyInfo[11],(BYTE*)&pCD->fParam0);
	 pT->GetRealParam(pT,&pMsg->m_sbyInfo[15],(BYTE*)&pCD->fParam1);
	 pT->GetRealParam(pT,&pMsg->m_sbyInfo[19],(BYTE*)&pCD->fParam2);
     return TRUE;
}
BOOL CDevice_EventHandler(This,SMESSAGE *pMsg)
{
	 DECLARE_SINGLE_OPEN(CDevice)
	 return TRUE;
}
BOOL CDevice_SaveChange(This,BYTE byEvent,WORD wValue,BOOL blAlarm)
{
    DECLARE_SINGLE_OPEN(CDevice)
}
BOOL CDevice_SavePinState(This,BYTE byEvent,WORD wValue)
{
    DECLARE_SINGLE_OPEN(CDevice)
}
void CDevice_SendSMessage(This,BYTE byBox,BYTE byFor,BYTE byType)
{
    DECLARE_SINGLE_OPEN(CDevice)
    SHORTMESSAGE m_sMsg;
	m_sMsg.m_swLen        = 9;
	m_sMsg.m_sbyFrom      = DIR_PHMDL;
	m_sMsg.m_sbyFor       = byFor;
	m_sMsg.m_sbyIntType   = 0;
	m_sMsg.m_sbyServerID  = 0;
	m_sMsg.m_sbyType      = byType;
	m_sMsg.m_sbyDirection = 0;
	m_sMsg.m_sbySensor    = 0;
	FPUT(byBox,(BYTE*)&m_sMsg);
    #ifdef DEB_CDevice
	Info("\n(__)CTLSN::>OUTT::%M",&m_sMsg);
    #endif
}
void CDevice_SendBroadcast(This,SKPEVENT *pEV)
{
}
void CDevice_SetInPinEvent(This)
{
    DECLARE_SINGLE_OPEN(CDevice)
}
void CDevice_SaveAlarmPin(This)
{
    DECLARE_SINGLE_OPEN(CDevice)
}
void CDevice_SendObsrveMsg(This)
{
    DECLARE_SINGLE_OPEN(CDevice)
}
PVOID CDevice_GetData(This,BYTE *pData,WORD *nLen)
{
    DECLARE_SINGLE_OPEN(CDevice)
}
WORD CDevice_GetWordParam(This,BYTE *pbyParam,BYTE *pbyOut)
{
    DECLARE_SINGLE_OPEN(CDevice)
	WORD wRes;
	#ifndef WIN32
	pbyOut[0] = pbyParam[1];
	pbyOut[1] = pbyParam[0];
    #else
	pbyOut[0] = pbyParam[0];
	pbyOut[1] = pbyParam[1];
    #endif
	memcpy(&wRes,&pbyOut[0],2);
	return wRes;
	//return (WORD)*((WORD*)pbyOut);
}
UDINT CDevice_GetDWordParam(This,BYTE *pbyParam,BYTE *pbyOut)
{
    DECLARE_SINGLE_OPEN(CDevice)
	DWORD wRes;
    #ifndef WIN32
	 pbyOut[3] = pbyParam[0];
	 pbyOut[2] = pbyParam[1];
	 pbyOut[1] = pbyParam[2];
	 pbyOut[0] = pbyParam[3];
    #else
	 memcpy(pbyOut,pbyParam,4);
    #endif
	memcpy(&wRes,&pbyOut[0],4);
	return wRes;
	//return (DWORD)*((DWORD*)pbyOut);
}
REAL CDevice_GetRealParam(This,BYTE *pbyParam,BYTE *pbyOut)
{
    DECLARE_SINGLE_OPEN(CDevice)
	REAL wRes;
    #ifndef WIN32
	pbyOut[3] = pbyParam[0];
	pbyOut[2] = pbyParam[1];
	pbyOut[1] = pbyParam[2];
	pbyOut[0] = pbyParam[3];
    #else
	memcpy(pbyOut,pbyParam,4);
	#endif
	memcpy(&wRes,&pbyOut[0],4);
	return wRes;
	//return (REAL)*((REAL*)pbyOut);
}
void CDevice_CDevice(This)
{
     DECLARE_SINGLE_OPEN(CDevice)
	 DECLARE_REGISTRATION(CDevice,Init)
	 //DECLARE_REGISTRATION(CDevice,GetW)
	 DECLARE_REGISTRATION(CDevice,SendSMessage)
	 DECLARE_REGISTRATION(CDevice,ObserveProc)
	 DECLARE_REGISTRATION(CDevice,PreProc)
	 DECLARE_REGISTRATION(CDevice,Processing)
	 DECLARE_REGISTRATION(CDevice,PostProc)
	 DECLARE_REGISTRATION(CDevice,SEventHandler)
	 DECLARE_REGISTRATION(CDevice,EventHandler)
	 DECLARE_REGISTRATION(CDevice,SaveChange)
	 DECLARE_REGISTRATION(CDevice,SavePinState)
	 DECLARE_REGISTRATION(CDevice,SendBroadcast)
	 DECLARE_REGISTRATION(CDevice,CheckAlarm)
	 DECLARE_REGISTRATION(CDevice,Switch)
	 DECLARE_REGISTRATION(CDevice,SetInPinEvent)
	 DECLARE_REGISTRATION(CDevice,SaveAlarmPin)
	 DECLARE_REGISTRATION(CDevice,SendObsrveMsg)
	 //DECLARE_REGISTRATION(CDevice,GetData)
	 DECLARE_REGISTRATION(CDevice,GetDWordParam)
	 DECLARE_REGISTRATION(CDevice,GetWordParam)
	 DECLARE_REGISTRATION(CDevice,GetRealParam)
	 DECLARE_REGISTRATION(CDevice,ExtractCMD)
	 /////////////////////////
	 DECLARE_REGISTRATION(CDevice,SetMsgAuto)
	 DECLARE_REGISTRATION(CDevice,GetStateList)
	 DECLARE_REGISTRATION(CDevice,HandleTask)
	 DECLARE_REGISTRATION(CDevice,HandleEvent)
	 DECLARE_REGISTRATION(CDevice,SetState)
	 DECLARE_REGISTRATION(CDevice,GetStateCode)
	 DECLARE_REGISTRATION(CDevice,GetState)
}
void CDevice_DCDevice(This)
{
	 DECLARE_SINGLE_OPEN(CDevice)
}
DECLARE_SINGLE_CREATE(CDevice)
```

#### bnrcount.h
```c
/********************************************************************
 * COPYRIGHT -- Kontora
 ********************************************************************
 * Program: bnrmain
 * File: bnraninput.h
 * Author: Abramenya
 * Created: January 19, 2009
 *******************************************************************/

#ifndef __COUNT_H__
#define __COUNT_H__
#include "typedefs.h"
#include "bnrdevice.h"
#include "bnrpin.h"

Class CCount
{
	 void (*CCCount)(This);
	 void (*DCCount)(This);
Public
     BYTE (*CheckTS)(This);
	 Virtual BOOL (*EventHandler)(This,SMESSAGE *pMsg);
	 Virtual void (*InitTCHN)(This,PVOID psTable);
     Virtual void (*PreProc)(This);
	 Virtual void (*Processing)(This);
     Virtual void (*PostProc)(This);
	 Virtual void (*SetInPinEvent)(This);
	 Virtual void (*SaveAlarmPin)(This);
	 Virtual void (*SendObsrveMsg)(This);
	 Virtual PVOID (*GetData)(This,BYTE *pData,WORD *nLen);
Public
     STCPARAM *pP;
	 DECLARE_IMPLEMENT_BASE(CDevice)
}
DECLARE_DEFINITION(CCount)
#endif
```

#### bnrcount.c
```c
/********************************************************************
 * COPYRIGHT -- Kontora
 ********************************************************************
 * Program: bnrmain
 * File: bnrlsens.c
 * Author: Abramenya
 * Created: January 19, 2009
 *******************************************************************/

#include "bnrcount.h"
#include "bnrmain.h"
#ifdef _DEFAULT_INCLUDES
 #include <AsDefault.h>
#endif
_GLOBAL BYTE nFSignal;
void CCount_InitTCHN(This,PVOID psTable)
{
    DECLARE_MULTI_OPEN(CCount,CDevice)
	pT->pP = (STCPARAM*)psTable;
	pB->m_nSize = sizeof(REAL)+sizeof(DWORD);
    #ifdef DEB_CCount
	//Info("\n(%b)CTLSG::>Create TeleSignal.",&pB->m_byID);
    #endif
}
void CCount_PreProc(This)
{
    DECLARE_MULTI_OPEN(CCount,CDevice)

}
_GLOBAL INT nTSCH;
void CCount_Processing(This)
{
	DECLARE_MULTI_OPEN(CCount,CDevice)
}
void CCount_PostProc(This)
{
	DECLARE_MULTI_OPEN(CCount,CDevice)
}
BYTE CCount_CheckTS(This)
{
    DECLARE_MULTI_OPEN(CCount,CDevice)
	//return pB->m_pPN->GetState(pB->m_pPN);
	return 0;
}
BOOL CCount_EventHandler(This,SMESSAGE *pMsg)
{
    DECLARE_MULTI_OPEN(CCount,CDevice)
    #ifdef DEB_CCount
	Info("\n(%b)CTLSG::>INPT::%M",&pB->m_nCD.wDeviceID,pMsg);
    #endif
	switch(pMsg->m_sbyFor)
	{
	  case DIR_MSTODV:
		   switch(pMsg->m_sbyType)
		   {
		    case PL_DATA_IND:
				 switch(pB->m_nCD.byParam0)
				 {
				   case CTR_TR:
                        //#ifdef DEB_CCount
	                    //Info("\n(%b)CTLSG::>CTR_TR::%d",&pB->m_nCD.wDeviceID,&pB->m_nCD.fParam0);
                        //#endif
						pT->pP->sDT.fKoeff = pB->m_nCD.fParam0;
				   break;
				   default:
				   break;
				 }
		    break;
			default:
            break;
		   }
      break;
	  case DIR_101MD:
	  break;
	  default:
	  break;
	}
	return TRUE;
}
void CCount_SetInPinEvent(This)
{
    DECLARE_MULTI_OPEN(CCount,CDevice)
}
void CCount_SaveAlarmPin(This)
{
	DECLARE_MULTI_OPEN(CCount,CDevice)
}
void CCount_SendObsrveMsg(This)
{
    DECLARE_MULTI_OPEN(CCount,CDevice)
}
/*
typedef struct _tagTCData
{
	REAL fKoeff;
	DWORD dwParam;
}STCDATA;
*/
PVOID CCount_GetData(This,BYTE *pData,WORD *nLen)
{
    DECLARE_MULTI_OPEN(CCount,CDevice)
	pB->GetRealParam(pB,(BYTE*)&pT->pP->sDT.fKoeff,pData);
	pB->GetDWordParam(pB,(BYTE*)&pT->pP->sDT.dwParam,&pData[4]);
	*nLen += pB->m_nSize;if (*nLen>350) *nLen=0;
	return pData;
}
void CCount_CCount(This)
{
    DECLARE_MULTI_OPEN(CCount,CDevice)
	DECLARE_REGISTRATION(CCount,CheckTS)
	DECLARE_VIRTUAL_FUNC(CCount,EventHandler)
	DECLARE_VIRTUAL_FUNC(CCount,InitTCHN)
	DECLARE_VIRTUAL_FUNC(CCount,PreProc)
	DECLARE_VIRTUAL_FUNC(CCount,Processing)
	DECLARE_VIRTUAL_FUNC(CCount,PostProc)
	DECLARE_VIRTUAL_FUNC(CCount,SetInPinEvent)
	DECLARE_VIRTUAL_FUNC(CCount,SaveAlarmPin)
	DECLARE_VIRTUAL_FUNC(CCount,SendObsrveMsg)
	DECLARE_VIRTUAL_FUNC(CCount,GetData)
}
void CCount_DCCount(This)
{
	DECLARE_MULTI_OPEN(CCount,CDevice)
}
DECLARE_MULTI_CREATE(CCount,CDevice)
```

#### AsTCP1.h - not listed in the package file held
```c
/* Automation Studio generated header file */
/* Do not edit ! */

#ifndef _ASTCP_
#define _ASTCP_

//#include <bur/plctypes.h>

//#include <runtime.h>

#ifndef _IEC_CONST
#define _IEC_CONST _WEAK const
#endif

/* Constants */
#ifdef _REPLACE_CONST
 #define tcpINVALID_IDENT 0U
 #define tcpSHUT_WR 2U
 #define tcpSHUT_RD 1U
 #define tcpOPT_REUSEADDR 1U
 #define tcpMSG_DONTROUTE 4U
 #define tcpMSG_PEEK 2U
 #define tcpMSG_OOB 1U
 #define tcpID_MAX_GET 3002U
 #define tcpID_LIST_GET 3001U
 #define tcpTCP_NODELAY_GET 2002U
 #define tcpTCP_NODELAY_SET 2001U
 #define tcpSO_ADDRESS_GET 1011U
 #define tcpSO_OOBINLINE_GET 1010U
 #define tcpSO_OOBINLINE_SET 1009U
 #define tcpSO_RCVBUF_GET 1008U
 #define tcpSO_RCVBUF_SET 1007U
 #define tcpSO_SNDBUF_GET 1006U
 #define tcpSO_SNDBUF_SET 1005U
 #define tcpSO_KEEPALIVE_GET 1004U
 #define tcpSO_KEEPALIVE_SET 1003U
 #define tcpSO_LINGER_GET 1002U
 #define tcpSO_LINGER_SET 1001U
 #define tcpERR_SYSTEM 32699U
 #define tcpERR_SOCKET_ACCEPT 32653U
 #define tcpERR_SOCKET_LISTEN 32652U
 #define tcpERR_SOCKET_BIND 32651U
 #define tcpERR_SOCKET_CREATE 32650U
 #define tcpERR_INTERFACE 32612U
 #define tcpERR_NO_OOBDATA 32611U
 #define tcpERR_ALREADY_CONNECTED 32610U
 #define tcpERR_NOT_CONNECTED 32609U
 #define tcpERR_INVALID 32608U
 #define tcpERR_WOULDBLOCK 32607U
 #define tcpERR_SENTLEN 32606U
 #define tcpERR_NO_DATA 32605U
 #define tcpERR_INVALID_IOCTL 32604U
 #define tcpERR_PARAMETER 32603U
 #define tcpERR_ALREADY_EXIST 32602U
 #define tcpERR_NOMORE_IDENTS 32601U
 #define tcpERR_INVALID_IDENT 32600U
#else
/*
 _IEC_CONST unsigned long tcpINVALID_IDENT = 0U;
 _IEC_CONST unsigned long tcpSHUT_WR = 2U;
 _IEC_CONST unsigned long tcpSHUT_RD = 1U;
 _IEC_CONST unsigned long tcpOPT_REUSEADDR = 1U;
 _IEC_CONST unsigned long tcpMSG_DONTROUTE = 4U;
 _IEC_CONST unsigned long tcpMSG_PEEK = 2U;
 _IEC_CONST unsigned long tcpMSG_OOB = 1U;
 _IEC_CONST unsigned long tcpID_MAX_GET = 3002U;
 _IEC_CONST unsigned long tcpID_LIST_GET = 3001U;
 _IEC_CONST unsigned long tcpTCP_NODELAY_GET = 2002U;
 _IEC_CONST unsigned long tcpTCP_NODELAY_SET = 2001U;
 _IEC_CONST unsigned long tcpSO_ADDRESS_GET = 1011U;
 _IEC_CONST unsigned long tcpSO_OOBINLINE_GET = 1010U;
 _IEC_CONST unsigned long tcpSO_OOBINLINE_SET = 1009U;
 _IEC_CONST unsigned long tcpSO_RCVBUF_GET = 1008U;
 _IEC_CONST unsigned long tcpSO_RCVBUF_SET = 1007U;
 _IEC_CONST unsigned long tcpSO_SNDBUF_GET = 1006U;
 _IEC_CONST unsigned long tcpSO_SNDBUF_SET = 1005U;
 _IEC_CONST unsigned long tcpSO_KEEPALIVE_GET = 1004U;
 _IEC_CONST unsigned long tcpSO_KEEPALIVE_SET = 1003U;
 _IEC_CONST unsigned long tcpSO_LINGER_GET = 1002U;
 _IEC_CONST unsigned long tcpSO_LINGER_SET = 1001U;
 _IEC_CONST unsigned short tcpERR_SYSTEM = 32699U;
 _IEC_CONST unsigned short tcpERR_SOCKET_ACCEPT = 32653U;
 _IEC_CONST unsigned short tcpERR_SOCKET_LISTEN = 32652U;
 _IEC_CONST unsigned short tcpERR_SOCKET_BIND = 32651U;
 _IEC_CONST unsigned short tcpERR_SOCKET_CREATE = 32650U;
 _IEC_CONST unsigned short tcpERR_INTERFACE = 32612U;
 _IEC_CONST unsigned short tcpERR_NO_OOBDATA = 32611U;
 _IEC_CONST unsigned short tcpERR_ALREADY_CONNECTED = 32610U;
 _IEC_CONST unsigned short tcpERR_NOT_CONNECTED = 32609U;
 _IEC_CONST unsigned short tcpERR_INVALID = 32608U;
 _IEC_CONST unsigned short tcpERR_WOULDBLOCK = 32607U;
 _IEC_CONST unsigned short tcpERR_SENTLEN = 32606U;
 _IEC_CONST unsigned short tcpERR_NO_DATA = 32605U;
 _IEC_CONST unsigned short tcpERR_INVALID_IOCTL = 32604U;
 _IEC_CONST unsigned short tcpERR_PARAMETER = 32603U;
 _IEC_CONST unsigned short tcpERR_ALREADY_EXIST = 32602U;
 _IEC_CONST unsigned short tcpERR_NOMORE_IDENTS = 32601U;
 _IEC_CONST unsigned short tcpERR_INVALID_IDENT = 32600U;
 */
#endif

/* Variables */

/* Datatypes and datatypes of function blocks */
typedef struct tcpLINGER_typ
{
	unsigned long lOnOff;
	unsigned long lLinger;
} tcpLINGER_typ;

typedef struct tcpSO_ADDRESS_typ
{
	unsigned long pPort;
	unsigned long pIpAddr;
} tcpSO_ADDRESS_typ;

typedef struct TcpOpen
{
	/* VAR_INPUT (analog) */
	unsigned long pIfAddr;
	unsigned short port;
	unsigned long options;
	/* VAR_OUTPUT (analog) */
	unsigned short status;
	unsigned long ident;
	/* VAR (analog) */
	unsigned short i_state;
	unsigned short i_result;
	unsigned long i_tmp;
        SOCKET sListen;
        SOCKET sClient;

	/* VAR_INPUT (digital) */
	BOOL enable;
} TcpOpen_typ;

typedef struct TcpServer
{
	/* VAR_INPUT (analog) */
	unsigned long ident;
	unsigned long backlog;
	unsigned long pIpAddr;
	/* VAR_OUTPUT (analog) */
	unsigned short status;
	unsigned long identclnt;
	unsigned short portclnt;
	/* VAR (analog) */
	unsigned short i_state;
	unsigned short i_result;
	unsigned long i_tmp;
	/* VAR_INPUT (digital) */
	BOOL enable;
} TcpServer_typ;

typedef struct TcpClient
{
	/* VAR_INPUT (analog) */
	unsigned long ident;
	unsigned long pServer;
	unsigned short portserv;
	/* VAR_OUTPUT (analog) */
	unsigned short status;
	/* VAR (analog) */
	unsigned short i_state;
	unsigned short i_result;
	unsigned long i_tmp;
	/* VAR_INPUT (digital) */
	BOOL enable;
} TcpClient_typ;

typedef struct TcpClose
{
	/* VAR_INPUT (analog) */
	unsigned long ident;
	unsigned long how;
	/* VAR_OUTPUT (analog) */
	unsigned short status;
	/* VAR (analog) */
	unsigned short i_state;
	unsigned short i_result;
	unsigned long i_tmp;
	/* VAR_INPUT (digital) */
	BOOL enable;
} TcpClose_typ;

typedef struct TcpSend
{
	/* VAR_INPUT (analog) */
	unsigned long ident;
	unsigned long pData;
	unsigned long datalen;
	unsigned long flags;
	/* VAR_OUTPUT (analog) */
	unsigned short status;
	unsigned long sentlen;
	/* VAR (analog) */
	unsigned short i_state;
	unsigned short i_result;
	unsigned long i_tmp;
	/* VAR_INPUT (digital) */
	BOOL enable;
} TcpSend_typ;

typedef struct TcpRecv
{
	/* VAR_INPUT (analog) */
	unsigned long ident;
	unsigned long pData;
	unsigned long datamax;
	unsigned long flags;
	/* VAR_OUTPUT (analog) */
	unsigned short status;
	unsigned long recvlen;
	/* VAR (analog) */
	unsigned short i_state;
	unsigned short i_result;
	unsigned long i_tmp;
	/* VAR_INPUT (digital) */
	BOOL enable;
} TcpRecv_typ;

typedef struct TcpIoctl
{
	/* VAR_INPUT (analog) */
	unsigned long ident;
	unsigned long ioctl;
	unsigned long pData;
	unsigned long datalen;
	/* VAR_OUTPUT (analog) */
	unsigned short status;
	unsigned long outlen;
	/* VAR (analog) */
	unsigned short i_state;
	unsigned short i_result;
	unsigned long i_tmp;
	/* VAR_INPUT (digital) */
	BOOL enable;
} TcpIoctl_typ;

/* Prototyping of functions and function blocks */
void TcpOpen(struct TcpOpen* inst);
void TcpServer(struct TcpServer* inst);
void TcpClient(struct TcpClient* inst);
void TcpClose(struct TcpClose* inst);
void TcpSend(struct TcpSend* inst);
void TcpRecv(struct TcpRecv* inst);
void TcpIoctl(struct TcpIoctl* inst);

#endif /* _ASTCP_ */
```

#### AsUDP1.h - not listed in the package file held
```c
/* Automation Studio generated header file */
/* Do not edit ! */

#ifndef _ASUDP_
#define _ASUDP_

//#include <bur/plctypes.h>

//#include <runtime.h>

#ifndef _IEC_CONST
#define _IEC_CONST _WEAK const
#endif

/* Constants */
#ifdef _REPLACE_CONST
 #define udpINVALID_IDENT 0U
 #define udpIP_TOS_MINCOST 2U
 #define udpIP_TOS_RELIABILITY 4U
 #define udpIP_TOS_THROUGHPUT 8U
 #define udpIP_TOS_LOWDELAY 16U
 #define udpOPT_BROADCAST 4U
 #define udpOPT_REUSEPORT 2U
 #define udpOPT_REUSEADDR 1U
 #define udpMSG_DONTROUTE 2U
 #define udpMSG_PEEK 1U
 #define udpID_MAX_GET 3002U
 #define udpID_LIST_GET 3001U
 #define udpIP_TTL_GET 2012U
 #define udpIP_TTL_SET 2011U
 #define udpIP_TOS_GET 2010U
 #define udpIP_TOS_SET 2009U
 #define udpIP_MULTICAST_LOOP_GET 2008U
 #define udpIP_MULTICAST_LOOP_SET 2007U
 #define udpIP_MULTICAST_TTL_GET 2006U
 #define udpIP_MULTICAST_TTL_SET 2005U
 #define udpIP_MULTICAST_IF_GET 2004U
 #define udpIP_MULTICAST_IF_SET 2003U
 #define udpIP_DROP_MEMBERSHIP 2002U
 #define udpIP_ADD_MEMBERSHIP 2001U
 #define udpSO_ADDRESS_GET 1007U
 #define udpSO_RCVBUF_GET 1006U
 #define udpSO_RCVBUF_SET 1005U
 #define udpSO_SNDBUF_GET 1004U
 #define udpSO_SNDBUF_SET 1003U
 #define udpSO_BROADCAST_GET 1002U
 #define udpSO_BROADCAST_SET 1001U
 #define udpERR_SYSTEM 32599U
 #define udpERR_SOCKET_CONNECT 32552U
 #define udpERR_SOCKET_BIND 32551U
 #define udpERR_SOCKET_CREATE 32550U
 #define udpERR_INTERFACE 32511U
 #define udpERR_UNREACHABLE 32510U
 #define udpERR_ACCESS 32509U
 #define udpERR_CONNREFUSED 32508U
 #define udpERR_WOULDBLOCK 32507U
 #define udpERR_SENTLEN 32506U
 #define udpERR_NO_DATA 32505U
 #define udpERR_INVALID_IOCTL 32504U
 #define udpERR_PARAMETER 32503U
 #define udpERR_ALREADY_EXIST 32502U
 #define udpERR_NOMORE_IDENTS 32501U
 #define udpERR_INVALID_IDENT 32500U
#else
/*
 _IEC_CONST unsigned long udpINVALID_IDENT = 0U;
 _IEC_CONST unsigned long udpIP_TOS_MINCOST = 2U;
 _IEC_CONST unsigned long udpIP_TOS_RELIABILITY = 4U;
 _IEC_CONST unsigned long udpIP_TOS_THROUGHPUT = 8U;
 _IEC_CONST unsigned long udpIP_TOS_LOWDELAY = 16U;
 _IEC_CONST unsigned long udpOPT_BROADCAST = 4U;
 _IEC_CONST unsigned long udpOPT_REUSEPORT = 2U;
 _IEC_CONST unsigned long udpOPT_REUSEADDR = 1U;
 _IEC_CONST unsigned long udpMSG_DONTROUTE = 2U;
 _IEC_CONST unsigned long udpMSG_PEEK = 1U;
 _IEC_CONST unsigned long udpID_MAX_GET = 3002U;
 _IEC_CONST unsigned long udpID_LIST_GET = 3001U;
 _IEC_CONST unsigned long udpIP_TTL_GET = 2012U;
 _IEC_CONST unsigned long udpIP_TTL_SET = 2011U;
 _IEC_CONST unsigned long udpIP_TOS_GET = 2010U;
 _IEC_CONST unsigned long udpIP_TOS_SET = 2009U;
 _IEC_CONST unsigned long udpIP_MULTICAST_LOOP_GET = 2008U;
 _IEC_CONST unsigned long udpIP_MULTICAST_LOOP_SET = 2007U;
 _IEC_CONST unsigned long udpIP_MULTICAST_TTL_GET = 2006U;
 _IEC_CONST unsigned long udpIP_MULTICAST_TTL_SET = 2005U;
 _IEC_CONST unsigned long udpIP_MULTICAST_IF_GET = 2004U;
 _IEC_CONST unsigned long udpIP_MULTICAST_IF_SET = 2003U;
 _IEC_CONST unsigned long udpIP_DROP_MEMBERSHIP = 2002U;
 _IEC_CONST unsigned long udpIP_ADD_MEMBERSHIP = 2001U;
 _IEC_CONST unsigned long udpSO_ADDRESS_GET = 1007U;
 _IEC_CONST unsigned long udpSO_RCVBUF_GET = 1006U;
 _IEC_CONST unsigned long udpSO_RCVBUF_SET = 1005U;
 _IEC_CONST unsigned long udpSO_SNDBUF_GET = 1004U;
 _IEC_CONST unsigned long udpSO_SNDBUF_SET = 1003U;
 _IEC_CONST unsigned long udpSO_BROADCAST_GET = 1002U;
 _IEC_CONST unsigned long udpSO_BROADCAST_SET = 1001U;
 _IEC_CONST unsigned short udpERR_SYSTEM = 32599U;
 _IEC_CONST unsigned short udpERR_SOCKET_CONNECT = 32552U;
 _IEC_CONST unsigned short udpERR_SOCKET_BIND = 32551U;
 _IEC_CONST unsigned short udpERR_SOCKET_CREATE = 32550U;
 _IEC_CONST unsigned short udpERR_INTERFACE = 32511U;
 _IEC_CONST unsigned short udpERR_UNREACHABLE = 32510U;
 _IEC_CONST unsigned short udpERR_ACCESS = 32509U;
 _IEC_CONST unsigned short udpERR_CONNREFUSED = 32508U;
 _IEC_CONST unsigned short udpERR_WOULDBLOCK = 32507U;
 _IEC_CONST unsigned short udpERR_SENTLEN = 32506U;
 _IEC_CONST unsigned short udpERR_NO_DATA = 32505U;
 _IEC_CONST unsigned short udpERR_INVALID_IOCTL = 32504U;
 _IEC_CONST unsigned short udpERR_PARAMETER = 32503U;
 _IEC_CONST unsigned short udpERR_ALREADY_EXIST = 32502U;
 _IEC_CONST unsigned short udpERR_NOMORE_IDENTS = 32501U;
 _IEC_CONST unsigned short udpERR_INVALID_IDENT = 32500U;
 */
#endif

/* Variables */

/* Datatypes and datatypes of function blocks */
typedef struct udpIP_MREQ_typ
{
	unsigned long pMcastAddr;
	unsigned long pIfAddr;
} udpIP_MREQ_typ;

typedef struct udpSO_ADDRESS_typ
{
	unsigned long pPort;
	unsigned long pIpAddr;
} udpSO_ADDRESS_typ;

typedef struct UdpOpen
{
	/* VAR_INPUT (analog) */
	unsigned long pIfAddr;
	unsigned short port;
	unsigned long options;
	/* VAR_OUTPUT (analog) */
	unsigned short status;
	unsigned long ident;
	/* VAR (analog) */
	unsigned short i_state;
	unsigned short i_result;
	unsigned long i_tmp;
	/* VAR_INPUT (digital) */
	BOOL enable;
} UdpOpen_typ;

typedef struct UdpClose
{
	/* VAR_INPUT (analog) */
	unsigned long ident;
	/* VAR_OUTPUT (analog) */
	unsigned short status;
	/* VAR (analog) */
	unsigned short i_state;
	unsigned short i_result;
	unsigned long i_tmp;
	/* VAR_INPUT (digital) */
	BOOL enable;
} UdpClose_typ;

typedef struct UdpConnect
{
	/* VAR_INPUT (analog) */
	unsigned long ident;
	unsigned long pHost;
	unsigned short port;
	/* VAR_OUTPUT (analog) */
	unsigned short status;
	/* VAR (analog) */
	unsigned short i_state;
	unsigned short i_result;
	unsigned long i_tmp;
	/* VAR_INPUT (digital) */
	BOOL enable;
} UdpConnect_typ;

typedef struct UdpDisconnect
{
	/* VAR_INPUT (analog) */
	unsigned long ident;
	/* VAR_OUTPUT (analog) */
	unsigned short status;
	/* VAR (analog) */
	unsigned short i_state;
	unsigned short i_result;
	unsigned long i_tmp;
	/* VAR_INPUT (digital) */
	BOOL enable;
} UdpDisconnect_typ;

typedef struct UdpSend
{
	/* VAR_INPUT (analog) */
	unsigned long ident;
	unsigned long pHost;
	unsigned short port;
	unsigned long pData;
	unsigned long datalen;
	unsigned long flags;
	/* VAR_OUTPUT (analog) */
	unsigned short status;
	unsigned long sentlen;
	/* VAR (analog) */
	unsigned short i_state;
	unsigned short i_result;
	unsigned long i_tmp;
	/* VAR_INPUT (digital) */
	BOOL enable;
} UdpSend_typ;

typedef struct UdpRecv
{
	/* VAR_INPUT (analog) */
	unsigned long ident;
	unsigned long pData;
	unsigned long datamax;
	unsigned long flags;
	unsigned long pIpAddr;
	/* VAR_OUTPUT (analog) */
	unsigned short status;
	unsigned long recvlen;
	unsigned short port;
	/* VAR (analog) */
	unsigned short i_state;
	unsigned short i_result;
	unsigned long i_tmp;
	/* VAR_INPUT (digital) */
	BOOL enable;
} UdpRecv_typ;

typedef struct UdpIoctl
{
	/* VAR_INPUT (analog) */
	unsigned long ident;
	unsigned long ioctl;
	unsigned long pData;
	unsigned long datalen;
	/* VAR_OUTPUT (analog) */
	unsigned short status;
	unsigned long outlen;
	/* VAR (analog) */
	unsigned short i_state;
	unsigned short i_result;
	unsigned long i_tmp;
	/* VAR_INPUT (digital) */
	BOOL enable;
} UdpIoctl_typ;

/* Prototyping of functions and function blocks */
void UdpOpen(struct UdpOpen* inst);
void UdpClose(struct UdpClose* inst);
void UdpConnect(struct UdpConnect* inst);
void UdpDisconnect(struct UdpDisconnect* inst);
void UdpSend(struct UdpSend* inst);
void UdpRecv(struct UdpRecv* inst);
void UdpIoctl(struct UdpIoctl* inst);

#endif /* _ASUDP_ */
```

#### bnralarm.h - not listed in the package file held
```c
/********************************************************************
 * COPYRIGHT -- Kontora
 ********************************************************************
 * Program: bnrmain
 * File: bnraninput.h
 * Author: Abramenya
 * Created: January 19, 2009
 *******************************************************************/

#ifndef __TMCOUNTER_H__
#define __TMCOUNTER_H__
#include "typedefs.h"
#include "bnrdevice.h"
#include "bnrpin.h"

Class CTmCounter
{
	 void (*CCTmCounter)(This);
	 void (*DCTmCounter)(This);
Public
     BYTE (*CheckTS)(This);
	 Virtual BOOL (*EventHandler)(This,SMESSAGE *pMsg);
	 Virtual void (*InitTCHN)(This,PVOID psTable);
     Virtual void (*PreProc)(This);
	 Virtual void (*Processing)(This);
     Virtual void (*PostProc)(This);
	 Virtual void (*SetInPinEvent)(This);
	 Virtual void (*SaveAlarmPin)(This);
	 Virtual void (*SendObsrveMsg)(This);
	 Virtual PVOID (*GetData)(This,BYTE *pData,WORD *nLen);
Public
     STMPARAM *pP;
	 BOOL *m_pbIN;
	 DECLARE_IMPLEMENT_BASE(CDevice)
}
DECLARE_DEFINITION(CTmCounter)
#endif
```

#### bnrswitcher.h - not listed in the package file held
```c
/********************************************************************
 * COPYRIGHT -- Kontora
 ********************************************************************
 * Program: bnrmain
 * File: bnraninput.h
 * Author: Abramenya
 * Created: January 19, 2009
 *******************************************************************/

#ifndef __SWITCHER_H__
#define __SWITCHER_H__
#include "typedefs.h"
#include "bnrdevice.h"
#include "bnrpin.h"

Class CSwitcher
{
	 void (*CCSwitcher)(This);
	 void (*DCSwitcher)(This);
Public
     BYTE (*CheckTS)(This);
	 Virtual BOOL (*EventHandler)(This,SMESSAGE *pMsg);
	 Virtual void (*InitTCHN)(This,PVOID psTable);
     Virtual void (*PreProc)(This);
	 Virtual void (*Processing)(This);
     Virtual void (*PostProc)(This);
	 Virtual void (*SetInPinEvent)(This);
	 Virtual void (*SaveAlarmPin)(This);
	 Virtual void (*SendObsrveMsg)(This);
	 Virtual PVOID (*GetData)(This,BYTE *pData,WORD *nLen);
Public
     SPLPARAM *pP;
	 BOOL *m_pbIN;
	 DECLARE_IMPLEMENT_BASE(CDevice)
}
DECLARE_DEFINITION(CSwitcher)
#endif
```

#### bnrudpinfoserver.h - not listed in the package file held
```c
/********************************************************************
 * COPYRIGHT -- Kontora
 ********************************************************************
 * Program: bnrmain
 * File: bnraninput.h
 * Author: Abramenya
 * Created: January 19, 2009
 *******************************************************************/

#ifndef __UDPINFOSERVER_H__
#define __UDPINFOSERVER_H__
#include "typedefs.h"
#include "bnrmessage.h"
#include "bnrdebug.h"
#include "bnrpob.h"
#include "bnrcyclicsystem.h"
#ifdef WIN32
#include "AsUdp1.h"
#include "winsock.h"
#else
//#include <Ethernet.h>
#endif
Class CUdpInfoServer
{
	 void (*CCUdpInfoServer)(This);
	 void (*DCUdpInfoServer)(This);
Public
     //Connection Disconnection Procedure
     void (*Init)(This,SARMINTERFACE *pArm);
     BOOL (*SendMessage)(This,SMESSAGE *pMsg);
	 BOOL (*GetMessage)(This,SMESSAGE *pMsg);
Private
	 BOOL (*Open)(This);
	 BOOL (*Listen)(This);
	 BOOL (*Close)(This,UDINT uModule);
	 BOOL (*CloseSend)(This);
	 BOOL (*CloseRecc)(This);
	 BOOL (*CheckSend)(This);
	 void (*PostSend)(This);
	 BOOL (*PostGet)(This);
	 void (*WordXCHG)(This,SMESSAGE *pMsg);
	 BOOL (*CheckCRC)(This,BOOL,SMESSAGE *pMsg);
     void (*AddCRC)(This,BOOL,SMESSAGE *pMsg);
	 DWORD (*ClcCRC)(This,BOOL,SMESSAGE *pMsg);
	 void (*ReceiveThread)(This);
	 void (*SendThread)(This);
	 Virtual BOOL (*EventHandler)(This,SMESSAGE *pMsg);
     Virtual void (*CyclicProc)(This);
Private
     SARMINTERFACE *m_pArm;
     UdpOpen_typ m_npListen;
     UdpSend_typ m_npSend;
	 UdpRecv_typ m_npRecc;
     UdpClose_typ m_npClose;
     BOOL m_blSState;
	 BOOL m_blRState;
     DWORD m_dwAPortNumber;
	 DWORD m_dwBPortNumber;
     char m_stUdpAddr[50];
	 BYTE m_bSrvState;
	 BYTE m_bCliState;
	 BYTE m_byConnReq;
	 SMESSAGE m_sMsg;
	 SMESSAGE m_sMsg0;
	 CMTimer m_nConnTMR;
	 DECLARE_IMPLEMENT_BASE(CCyclicSystem)
}
DECLARE_DEFINITION(CUdpInfoServer)
#endif
```

#### Ethernet1.h - not listed in the package file held
```c
/* Automation Studio Generated Header File, Format Version 1.00 */
/* do not change */
#ifndef ETHERNET_H1_
#define ETHERNET_H1_

/* Datatypes */
typedef struct TCPQ_dcmd_typ
{
	unsigned short response;
	unsigned long error;
	unsigned long buffer;
	unsigned long buflng;
	unsigned long ipaddr;
	unsigned long socket;
	unsigned short port;
	unsigned short wreserve;
	unsigned long reserve[8];
} TCPQ_dcmd_typ;

typedef struct ETHstat_typ
{
	unsigned long l_int;
	unsigned long l_rint;
	unsigned long l_tint;
	unsigned short l_babl;
	unsigned short l_cerr;
	unsigned short l_miss;
	unsigned short l_memr;
	unsigned short r_fram;
	unsigned short r_oflo;
	unsigned short r_crc;
	unsigned short r_buff;
	unsigned short t_buff;
	unsigned short t_uflo;
	unsigned short t_lcol;
	unsigned short t_lcar;
	unsigned short t_rtry;
	unsigned short ni_anno;
	unsigned short ni_init;
	unsigned short ni_send;
	unsigned short ni_getp;
	unsigned short ni_retp;
	unsigned short ni_bcst;
	unsigned short ni_poll;
	unsigned short irq_mean;
	unsigned short irq_min;
	unsigned short irq_max;
	unsigned short irq_t1;
	unsigned short irq_timena;
	unsigned short errgtnobuf;
	unsigned short err_1_1;
	unsigned short err_1_2;
	unsigned short err_1_3;
	unsigned short errxmtnull;
	unsigned short errsndown;
	unsigned short errsndsize;
	unsigned short lancerrnobuf;
	unsigned short lanceinit;
	unsigned short terr;
	unsigned short ni_gtbuf;
	unsigned short brcast_cnt;
	unsigned short brcastmax_cnt;
	unsigned short brcast_stop;
	unsigned short brcast_tick;
} ETHstat_typ;

typedef struct ETHattachment_typ
{
	unsigned char type;
	unsigned long len;
	unsigned long pName;
	unsigned long pData;
} ETHattachment_typ;

/* Datatypes of function blocks */
typedef struct UDPsend
{
	/* VAR_INPUT (analogous) */
	unsigned long cident;
	unsigned long ipaddr;
	unsigned long buffer;
	unsigned short buflng;
	unsigned short port;
	/* VAR_OUTPUT (analogous) */
	unsigned short status;
	/* VAR (analogous) */
	unsigned short state;
	unsigned long tickcount;
	unsigned long initcount;
	struct TCPQ_dcmd_typ dcmd;
	/* VAR_INPUT (digital) */
	BOOL enable;
	/* VAR (digital) */
	BOOL pna_ok;
} UDPsend_typ;

typedef struct UDPrecv
{
	/* VAR_INPUT (analogous) */
	unsigned long cident;
	unsigned long buffer;
	unsigned short buflng;
	/* VAR_OUTPUT (analogous) */
	unsigned short status;
	unsigned long ipaddr;
	unsigned short rxbuflng;
	unsigned short port;
	/* VAR (analogous) */
	unsigned short state;
	unsigned long tickcount;
	unsigned long initcount;
	struct TCPQ_dcmd_typ dcmd;
	/* VAR_INPUT (digital) */
	BOOL enable;
	/* VAR (digital) */
	BOOL pna_ok;
} UDPrecv_typ;

typedef struct UDPopen
{
	/* VAR_INPUT (analogous) */
	unsigned short port;
	unsigned long pvpolladr;
	/* VAR_OUTPUT (analogous) */
	unsigned short status;
	unsigned long cident;
	/* VAR (analogous) */
	unsigned short state;
	unsigned long tickcount;
	unsigned long initcount;
	struct TCPQ_dcmd_typ dcmd;
	/* VAR_INPUT (digital) */
	BOOL enable;
	/* VAR (digital) */
	BOOL pna_ok;
} UDPopen_typ;

typedef struct UDPclose
{
	/* VAR_INPUT (analogous) */
	unsigned long cident;
	/* VAR_OUTPUT (analogous) */
	unsigned short status;
	/* VAR (analogous) */
	unsigned short state;
	unsigned long tickcount;
	unsigned long initcount;
	struct TCPQ_dcmd_typ dcmd;
	/* VAR_INPUT (digital) */
	BOOL enable;
	/* VAR (digital) */
	BOOL pna_ok;
} UDPclose_typ;

typedef struct ETHinfo
{
	/* VAR_OUTPUT (analogous) */
	unsigned long statadr;
	unsigned long ethadr;
	unsigned short status;
	/* VAR (analogous) */
	unsigned long address1;
	unsigned long address2;
	/* VAR_INPUT (digital) */
	BOOL enable;
} ETHinfo_typ;

typedef struct ETHnode
{
	/* VAR_OUTPUT (analogous) */
	unsigned short status;
	unsigned char nodenr;
	unsigned long ipaddr;
	/* VAR (analogous) */
	unsigned long address1;
	unsigned long address2;
	/* VAR_INPUT (digital) */
	BOOL enable;
} ETHnode_typ;

typedef struct TCPserv
{
	/* VAR_INPUT (analogous) */
	unsigned short porta;
	/* VAR_OUTPUT (analogous) */
	unsigned short status;
	unsigned long ipaddr;
	unsigned short portb;
	unsigned long cident;
	/* VAR (analogous) */
	unsigned short state;
	unsigned long tickcount;
	unsigned long initcount;
	SOCKET  sListen;
	SOCKET  sClient;
	struct TCPQ_dcmd_typ dcmd;
	/* VAR_INPUT (digital) */
	BOOL enable;
	/* VAR (digital) */
	BOOL pna_ok;
} TCPserv_typ;

typedef struct TCPclient
{
	/* VAR_INPUT (analogous) */
	unsigned short porta;
	unsigned long ipaddr;
	unsigned short portb;
	/* VAR_OUTPUT (analogous) */
	unsigned short status;
	unsigned long cident;
	/* VAR (analogous) */
	unsigned short state;
	unsigned long tickcount;
	unsigned long initcount;
	struct TCPQ_dcmd_typ dcmd;
	/* VAR_INPUT (digital) */
	BOOL enable;
	/* VAR (digital) */
	BOOL pna_ok;
} TCPclient_typ;

typedef struct TCPsend
{
	/* VAR_INPUT (analogous) */
	unsigned long cident;
	unsigned long buffer;
	unsigned long buflng;
	/* VAR_OUTPUT (analogous) */
	unsigned short status;
	/* VAR (analogous) */
	unsigned short state;
	unsigned long tickcount;
	unsigned long initcount;
	struct TCPQ_dcmd_typ dcmd;
	/* VAR_INPUT (digital) */
	BOOL enable;
	/* VAR (digital) */
	BOOL pna_ok;
} TCPsend_typ;

typedef struct TCPrecv
{
	/* VAR_INPUT (analogous) */
	unsigned long cident;
	unsigned long buffer;
	unsigned long mxbuflng;
	/* VAR_OUTPUT (analogous) */
	unsigned short status;
	unsigned long rxbuflng;
	/* VAR (analogous) */
	unsigned short state;
	unsigned long tickcount;
	unsigned long initcount;
	struct TCPQ_dcmd_typ dcmd;
	/* VAR_INPUT (digital) */
	BOOL enable;
	/* VAR (digital) */
	BOOL pna_ok;
} TCPrecv_typ;

typedef struct TCPclose
{
	/* VAR_INPUT (analogous) */
	unsigned long cident;
	/* VAR_OUTPUT (analogous) */
	unsigned short status;
	/* VAR (analogous) */
	unsigned short state;
	unsigned long tickcount;
	unsigned long initcount;
	struct TCPQ_dcmd_typ dcmd;
	/* VAR_INPUT (digital) */
	BOOL enable;
	/* VAR (digital) */
	BOOL pna_ok;
} TCPclose_typ;

typedef struct SMTPxsendmail
{
	/* VAR_INPUT (analogous) */
	unsigned long pReceiver;
	unsigned long pSender;
	unsigned long pIpaddr;
	unsigned long pSubject;
	unsigned long pText;
	unsigned long pAttachment;
	unsigned char AttachmentCount;
	unsigned short timeout;
	/* VAR_OUTPUT (analogous) */
	unsigned short status;
	/* VAR (analogous) */
	unsigned short state;
	unsigned long tickcount;
	unsigned long initcount;
	struct TCPQ_dcmd_typ dcmd;
	/* VAR_INPUT (digital) */
	BOOL enable;
	/* VAR (digital) */
	BOOL pna_ok;
} SMTPxsendmail_typ;

typedef struct SMTPsendmail
{
	/* VAR_INPUT (analogous) */
	unsigned long pReceiver;
	unsigned long pSender;
	unsigned long pIpaddr;
	unsigned long pSubject;
	unsigned long pText;
	unsigned short timeout;
	/* VAR_OUTPUT (analogous) */
	unsigned short status;
	/* VAR (analogous) */
	unsigned short state;
	unsigned long tickcount;
	unsigned long initcount;
	struct TCPQ_dcmd_typ dcmd;
	/* VAR_INPUT (digital) */
	BOOL enable;
	/* VAR (digital) */
	BOOL pna_ok;
} SMTPsendmail_typ;

typedef struct ICMPping
{
	/* VAR_INPUT (analogous) */
	unsigned long ipaddr;
	unsigned short timeout;
	/* VAR_OUTPUT (analogous) */
	unsigned short status;
	/* VAR (analogous) */
	unsigned short state;
	unsigned long tickcount;
	unsigned long initcount;
	struct TCPQ_dcmd_typ dcmd;
	/* VAR_INPUT (digital) */
	BOOL enable;
	/* VAR (digital) */
	BOOL pna_ok;
} ICMPping_typ;

/* Prototyping of functions and function blocks */
void UDPsend(UDPsend_typ* inst);
void UDPrecv(UDPrecv_typ* inst);
void UDPopen(UDPopen_typ* inst);
void UDPclose(UDPclose_typ* inst);
void ETHinfo(ETHinfo_typ* inst);
void ETHnode(ETHnode_typ* inst);
void TCPserv(TCPserv_typ* inst);
void TCPclient(TCPclient_typ* inst);
void TCPsend(TCPsend_typ* inst);
void TCPrecv(TCPrecv_typ* inst);
void TCPclose(TCPclose_typ* inst);
void SMTPxsendmail(SMTPxsendmail_typ* inst);
void SMTPsendmail(SMTPsendmail_typ* inst);
void ICMPping(ICMPping_typ* inst);

#endif /* ETHERNET_H_ */
```

#### bnralarm.c - not listed in the package file held
```c
/********************************************************************
 * COPYRIGHT -- Kontora
 ********************************************************************
 * Program: bnrmain
 * File: bnrlsens.c
 * Author: Abramenya
 * Created: January 19, 2009
 *******************************************************************/

#include "bnrtmcounter.h"
#include "bnrmain.h"
#ifdef _DEFAULT_INCLUDES
 #include <AsDefault.h>
#endif
_GLOBAL BYTE nFSignal;
void CTmCounter_InitTCHN(This,PVOID psTable)
{
    DECLARE_MULTI_OPEN(CTmCounter,CDevice)
    pT->pP = (STMPARAM*)psTable;
	pB->m_nSize = 2*sizeof(WORD);
    #ifdef DEB_CTmCounter
	//Info("\n(%b)CTLSG::>Create TeleSignal.",&pB->m_byID);
    #endif
}
void CTmCounter_PreProc(This)
{
    DECLARE_MULTI_OPEN(CTmCounter,CDevice)

}
_GLOBAL INT nTSCH;
void CTmCounter_Processing(This)
{
	DECLARE_MULTI_OPEN(CTmCounter,CDevice)
}
void CTmCounter_PostProc(This)
{
	DECLARE_MULTI_OPEN(CTmCounter,CDevice)
	BOOL res = FALSE;
}
BYTE CTmCounter_CheckTS(This)
{
    DECLARE_MULTI_OPEN(CTmCounter,CDevice)
    //return pB->m_pPN->GetState(pB->m_pPN);
	return 0;
}
BOOL CTmCounter_EventHandler(This,SMESSAGE *pMsg)
{
    DECLARE_MULTI_OPEN(CTmCounter,CDevice)
    BYTE byID = pMsg->m_sbySensor;
	BYTE byParamType = pMsg->m_sbyInfo[3];
    #ifdef DEB_CTmCounter
	Info("\n(%b)CTLSG::>INPT::%M",&pB->m_byID,pMsg);
    #endif
	switch(pMsg->m_sbyFor)
	{
	  case DIR_101TOKP:
		   switch(pMsg->m_sbyType)
		   {
		    case PL_DATA_IND:
				 //Info("\n(%b)CTLSG::>DL_DATA_IND::>%M",&pB->m_byID,pMsg);
				 switch(byParamType)
				 {
				   case EN_SET_PERIOD:
					    //pT->m_byCSetPulce = pMsg->m_sbyInfo[3];
					    //pT->m_bySetPulce  = pT->m_byCSetPulce;
				   break;
				   case EN_REM_PERIOD:
					    //pT->m_byRemPulce  = pMsg->m_sbyInfo[3];
						//pT->m_byCRemPulce = pT->m_byRemPulce;
				   break;
				   case EN_PIN_ALMODE:
                        //pT->m_byAlarmMode = pMsg->m_sbyInfo[3];
				   break;
				   default:
				   break;
				 }
		    break;
			default:
            break;
		   }
      break;
	  case DIR_101MD:
	  break;
	  default:
	  break;
	}
	return TRUE;
}
void CTmCounter_SetInPinEvent(This)
{
    DECLARE_MULTI_OPEN(CTmCounter,CDevice)
}
void CTmCounter_SaveAlarmPin(This)
{
	DECLARE_MULTI_OPEN(CTmCounter,CDevice)
}
void CTmCounter_SendObsrveMsg(This)
{
    DECLARE_MULTI_OPEN(CTmCounter,CDevice)
}
/*
typedef struct _tagTTMData
{
UINT wJob;
UINT wParam;
}STTMDATA;
*/
PVOID CTmCounter_GetData(This,BYTE *pData,WORD *nLen)
{
    DECLARE_MULTI_OPEN(CTmCounter,CDevice)
	pB->GetWordParam(pB,(BYTE*)&pT->pP->sDT.wJob,&pData[0]);
	pB->GetWordParam(pB,(BYTE*)&pT->pP->sDT.wParam,&pData[2]);
	*nLen += pB->m_nSize;if (*nLen>350) *nLen=0;
	return pData;
}
void CTmCounter_CTmCounter(This)
{
    DECLARE_MULTI_OPEN(CTmCounter,CDevice)
	DECLARE_REGISTRATION(CTmCounter,CheckTS)
	DECLARE_VIRTUAL_FUNC(CTmCounter,EventHandler)
	DECLARE_VIRTUAL_FUNC(CTmCounter,InitTCHN)
	DECLARE_VIRTUAL_FUNC(CTmCounter,PreProc)
	DECLARE_VIRTUAL_FUNC(CTmCounter,Processing)
	DECLARE_VIRTUAL_FUNC(CTmCounter,PostProc)
	DECLARE_VIRTUAL_FUNC(CTmCounter,SetInPinEvent)
	DECLARE_VIRTUAL_FUNC(CTmCounter,SaveAlarmPin)
	DECLARE_VIRTUAL_FUNC(CTmCounter,SendObsrveMsg)
	DECLARE_VIRTUAL_FUNC(CTmCounter,GetData)
}
void CTmCounter_DCTmCounter(This)
{
	DECLARE_MULTI_OPEN(CTmCounter,CDevice)
}
DECLARE_MULTI_CREATE(CTmCounter,CDevice)
```

#### bnrswitcher.c - not listed in the package file held
```c
/********************************************************************
 * COPYRIGHT -- Kontora
 ********************************************************************
 * Program: bnrmain
 * File: bnrlsens.c
 * Author: Abramenya
 * Created: January 19, 2009
 *******************************************************************/

#include "bnrswitcher.h"
#include "bnrmain.h"
#ifdef _DEFAULT_INCLUDES
 #include <AsDefault.h>
#endif
_GLOBAL BYTE nFSignal;
void CSwitcher_InitTCHN(This,PVOID psTable)
{
    DECLARE_MULTI_OPEN(CSwitcher,CDevice)
    pT->pP = (SPLPARAM*)psTable;
	pB->m_nSize = 1;
    #ifdef DEB_CSwitcher
	//Info("\n(%b)CTLSG::>Create TeleSignal.",&pB->m_byID);
    #endif
}
void CSwitcher_PreProc(This)
{
    DECLARE_MULTI_OPEN(CSwitcher,CDevice)

}
_GLOBAL INT nTSCH;
void CSwitcher_Processing(This)
{
	DECLARE_MULTI_OPEN(CSwitcher,CDevice)
}
void CSwitcher_PostProc(This)
{
	DECLARE_MULTI_OPEN(CSwitcher,CDevice)
	BOOL res = FALSE;
}
BYTE CSwitcher_CheckTS(This)
{
    DECLARE_MULTI_OPEN(CSwitcher,CDevice)
    //return pB->m_pPN->GetState(pB->m_pPN);
	return 0;
}
BOOL CSwitcher_EventHandler(This,SMESSAGE *pMsg)
{
    DECLARE_MULTI_OPEN(CSwitcher,CDevice)
    BYTE byID = pMsg->m_sbySensor;
	BYTE byParamType = pMsg->m_sbyInfo[3];
    #ifdef DEB_CSwitcher
	Info("\n(%b)CTLSG::>INPT::%M",&pB->m_byID,pMsg);
    #endif
	switch(pMsg->m_sbyFor)
	{
	  case DIR_101TOKP:
		   switch(pMsg->m_sbyType)
		   {
		    case PL_DATA_IND:
				 //Info("\n(%b)CTLSG::>DL_DATA_IND::>%M",&pB->m_byID,pMsg);
				 switch(byParamType)
				 {
				   case EN_SET_PERIOD:
					    //pT->m_byCSetPulce = pMsg->m_sbyInfo[3];
					    //pT->m_bySetPulce  = pT->m_byCSetPulce;
				   break;
				   case EN_REM_PERIOD:
					    //pT->m_byRemPulce  = pMsg->m_sbyInfo[3];
						//pT->m_byCRemPulce = pT->m_byRemPulce;
				   break;
				   case EN_PIN_ALMODE:
                        //pT->m_byAlarmMode = pMsg->m_sbyInfo[3];
				   break;
				   default:
				   break;
				 }
		    break;
			default:
            break;
		   }
      break;
	  case DIR_101MD:
	  break;
	  default:
	  break;
	}
	return TRUE;
}
void CSwitcher_SetInPinEvent(This)
{
    DECLARE_MULTI_OPEN(CSwitcher,CDevice)
}
void CSwitcher_SaveAlarmPin(This)
{
	DECLARE_MULTI_OPEN(CSwitcher,CDevice)
}
void CSwitcher_SendObsrveMsg(This)
{
    DECLARE_MULTI_OPEN(CSwitcher,CDevice)
}
/*
typedef struct _tagTTMData
{
UINT wJob;
UINT wParam;
}STTMDATA;
*/
PVOID CSwitcher_GetData(This,BYTE *pData,WORD *nLen)
{
    DECLARE_MULTI_OPEN(CSwitcher,CDevice)
    pData[0] = pT->pP->sDT.byParam;
	*nLen += pB->m_nSize;if (*nLen>350) *nLen=0;
	return pData;
}
void CSwitcher_CSwitcher(This)
{
    DECLARE_MULTI_OPEN(CSwitcher,CDevice)
	DECLARE_REGISTRATION(CSwitcher,CheckTS)
	DECLARE_VIRTUAL_FUNC(CSwitcher,EventHandler)
	DECLARE_VIRTUAL_FUNC(CSwitcher,InitTCHN)
	DECLARE_VIRTUAL_FUNC(CSwitcher,PreProc)
	DECLARE_VIRTUAL_FUNC(CSwitcher,Processing)
	DECLARE_VIRTUAL_FUNC(CSwitcher,PostProc)
	DECLARE_VIRTUAL_FUNC(CSwitcher,SetInPinEvent)
	DECLARE_VIRTUAL_FUNC(CSwitcher,SaveAlarmPin)
	DECLARE_VIRTUAL_FUNC(CSwitcher,SendObsrveMsg)
	DECLARE_VIRTUAL_FUNC(CSwitcher,GetData)
}
void CSwitcher_DCSwitcher(This)
{
	DECLARE_MULTI_OPEN(CSwitcher,CDevice)
}
DECLARE_MULTI_CREATE(CSwitcher,CDevice)
```

#### bnrtcpserver0.c - not listed in the package file held
```c
/********************************************************************
 * COPYRIGHT -- Kontora
 ********************************************************************
 * Program: bnrmain
 * File: bnrlsens.c
 * Author: Abramenya
 * Created: January 19, 2009
 *******************************************************************/

#include "bnrtcpserver.h"
#ifdef _DEFAULT_INCLUDES
 #include <AsDefault.h>
#endif
_GLOBAL	 TcpServer_typ m_npServer[1];
_GLOBAL  TcpOpen_typ m_npListen[1];
_GLOBAL  TcpSend_typ m_npSend[1];
_GLOBAL	 TcpRecv_typ m_npRecc[1];
_GLOBAL  TcpClose_typ m_npClose[1];
#ifdef WIN32
DWORD dwThreadId;
//void TcpOpen(TcpOpen_typ *pServer){pServer->status=0;}
SOCKET sClient;
DWORD WINAPI GetArm(PVOID pVoid);
void TcpClose(TcpClose_typ *pCL){};
void TcpServer(TcpServer_typ *pServer){pServer->identclnt=pServer->ident;pServer->status=0;}
void TcpOpen(TcpOpen_typ *pServer)
{
	BOOL    bInterface = FALSE;
    WSADATA wsd;
	int iAddrSize;
	struct sockaddr_in local,client;
	struct sockaddr_in server;
    struct hostent *host = NULL;
	pServer->status = 1;
	if (WSAStartup(MAKEWORD(2,2), &wsd) != 0)
    {
        printf("Failed to load Winsock!\n");
        return ;
    }
	pServer->sListen = socket(AF_INET, SOCK_STREAM, IPPROTO_TCP);
    if (pServer->sListen == SOCKET_ERROR)
    {
        printf("socket() failed: %d\n", WSAGetLastError());
        return ;
    }
    if (bInterface)
    {
        //local.sin_addr.s_addr = inet_addr(pServer->pIfAddr);
		local.sin_addr.s_addr = inet_addr("0.0.0.0");
        if (local.sin_addr.s_addr == INADDR_NONE)
		{
			printf("socket() failed: %s\n", pServer->pIfAddr);
			return;
		}
    }
    else
		local.sin_addr.s_addr = htonl(INADDR_ANY);
	local.sin_family = AF_INET;
	local.sin_port = htons((u_short)pServer->port);
    if (bind(pServer->sListen, (struct sockaddr *)&local,sizeof(local)) == SOCKET_ERROR)
    {
        printf("bind() failed: %d\n", WSAGetLastError());
        return ;
    }
    listen(pServer->sListen, 8);
    iAddrSize = sizeof(client);
    //pServer->sClient = accept(pServer->sListen, (struct sockaddr *)&client,&iAddrSize);
	pServer->sClient = accept(pServer->sListen, (struct sockaddr *)&client,&iAddrSize);
    if (pServer->sClient == INVALID_SOCKET)
    {
		printf("accept() failed: %d\n", WSAGetLastError());
		return ;
    }
	sClient = pServer->sClient;
	pServer->ident = &pServer->sClient;
	Info("\n(__)CTCPS::>Connect");
	pServer->status = 0;
}
//void TcpSend(TcpSend_typ *pCL){};
void TcpSend(TcpSend_typ *pSend)
{
	int ret;
	ret = send(sClient, (char*)pSend->pData, pSend->datalen, 0);
	//Info("\n(__)ARM_0:%M",pSend->buffer);
	if (ret == 0)
	{
		//printf("Send Not Poss \n");
		//Sleep(500);
		pSend->status = 1;
		return;
	}
	else if (ret == SOCKET_ERROR)
	{
		//printf("send() failed: %d\n",WSAGetLastError());
		//Sleep(500);
		pSend->status = 1;
		return;
	}
	//Sleep(50);
	pSend->status = 0;

}
void TcpRecv(TcpRecv_typ *pRecv)
{
	int ret;
	//printf("RCV\n");
	ret = recv(sClient,(char*)pRecv->pData,pRecv->datamax , 0);
	if (ret == 0)
	{
		//Sleep(500);
		printf("recv() failed 0: %d\n", WSAGetLastError());
		pRecv->status = 1;
		return;
	}
	else if (ret == SOCKET_ERROR)
	{
		printf("recv() failed: %d\n", WSAGetLastError());
        //Sleep(500);
		pRecv->status = 1;
		return;
	}
	//printf("Reccive OK! \n");
	pRecv->recvlen = ret;
	pRecv->status = 0;
}
#endif

//_GLOBAL INT iCreate1;
_GLOBAL UINT iCreateTcp1;
void CTcpServer_Init(This,SARMINTERFACE *pArm)
{
    DECLARE_MULTI_OPEN(CTcpServer,CCyclicSystem)
	FDEFINE(DEV_TCPRM_BOX_ID,1024);
	FDEFINE(DEV_TCPBF_BOX_ID,1024);
	pB->SetBoxID(pB,DEV_TCPRM_BOX_ID);
	InitObject(CMTimer,&pT->m_nConnTMR);
	pT->m_nConnTMR.SetTimer(&pT->m_nConnTMR,DIR_TCPTOTCP,DIR_TCPTOTCP,EV_TMR_SRR_REQ,0,0,DEV_TCPRM_BOX_ID);
	pT->m_pArm = pArm;
	pT->m_dwAPortNumber = pArm->dwpPortNumber[0];
	pT->m_dwBPortNumber = pArm->dwpPortNumber[1];
	strcpy(pT->m_stTcpAddr,pArm->chTcpAddr);
	#ifdef DEB_CTcpServer
	Info("\n\r(__)CTcpS::>Create Tcp.PA: %d.PB: %d. Addr[%s]",&pT->m_dwAPortNumber,&pT->m_dwBPortNumber,pT->m_stTcpAddr);
    #endif
 	pT->m_npListen =  &m_npListen[0];
	pT->m_npSend   =  &m_npSend[0];
	pT->m_npRecc   =  &m_npRecc[0];
	pT->m_npClose  =  &m_npClose[0];
	pT->m_npServer =  &m_npServer[0];

	memset(pT->m_npListen,0,sizeof(TcpOpen_typ));
	//memset(pT->m_npSend,0,sizeof(TcpSend_typ));
	//memset(&pT->m_npRecc,0,sizeof(TcpRecv_typ));
	pT->m_npListen->enable  = TRUE;
	pT->m_npListen->port    = pT->m_dwAPortNumber;
	pT->m_npListen->pIfAddr = 0;
	pT->m_npListen->status  = 1;
	pT->m_npListen->options = 0;

	pT->m_blSState = TRUE;
	pT->m_blRState = TRUE;
	pT->m_bSrvState = DRV_ST_DISC;

	pT->m_nConnTMR.OnTimer(&pT->m_nConnTMR,100);
    #ifdef WIN32
	CreateThread(NULL,0,GetArm ,pT,0,&dwThreadId);
	#endif
}
_GLOBAL TcpServer_typ sServer;
_GLOBAL TcpRecv_typ sRecc;
BOOL CTcpServer_Open(This)
{
	DECLARE_MULTI_OPEN(CTcpServer,CCyclicSystem)

	if(pT->m_bSrvState==DRV_ST_DISC)
	{
	 if (pT->m_byConnReq++%2==0)
	 {
	  pT->CloseRecc(pT);
	  pT->CloseSend(pT);
	  pT->CloseOpen(pT);
	 }
	 pT->Listen(pT);
	}

	if(pT->m_bSrvState==DRV_ST_OPEN)
	{
	 //memset(pT->m_npServer,0,sizeof(TcpServer_typ));
	 pT->m_npServer->enable  = 1;
	 pT->m_npServer->ident   = pT->m_npListen->ident;
	 pT->m_npServer->backlog = 1;
	 pT->m_npServer->pIpAddr = pT->m_stTcpAddr;
     TcpServer(pT->m_npServer);
	 memcpy(&sServer,pT->m_npServer,sizeof(TcpServer_typ));
     if(pT->m_npServer->status==0)
	 {

	  //if(pT->m_bSrvState==DRV_ST_OPEN)
      pT->m_npRecc->enable   = 1;
      pT->m_npRecc->ident    = pT->m_npServer->identclnt;
	  pT->m_npRecc->datamax  = sizeof(SMESSAGE)-10;
	  pT->m_npRecc->flags     = 0;

	  pT->m_npSend->enable   = 1;
	  pT->m_npSend->ident    = pT->m_npServer->identclnt;
	  pT->m_npSend->datalen  = sizeof(SMESSAGE);
	  pT->m_npSend->flags    = 0;
	  pT->m_bSrvState = DRV_ST_CONN;
	  pT->m_blSState = TRUE;
	  //pT->Connect(pT);
	  //pT->SendSMessage(pT,DEV_KPMDL_BOX_ID,DIR_PHTOKP,PH_CALL_REQ);
  	  return TRUE;
	 }
	}
    return TRUE;
}
_GLOBAL TcpOpen_typ sOpen;
_GLOBAL INT iListen;
BOOL CTcpServer_Listen(This)
{
    DECLARE_MULTI_OPEN(CTcpServer,CCyclicSystem)
	iListen++;
	memset(pT->m_npListen,0,sizeof(TcpOpen_typ));
	pT->m_npListen->enable  = 1;
	pT->m_npListen->port    = pT->m_dwAPortNumber;
	pT->m_npListen->pIfAddr = 0;
	pT->m_npListen->status  = 1;
	pT->m_npListen->options = 0;
	//memcpy(&sOpen,pT->m_npListen,sizeof(TcpOpen_typ));
    TcpOpen(pT->m_npListen);
	//TcpOpen(&sOpen);
 	memcpy(&sOpen,pT->m_npListen,sizeof(TcpOpen_typ));
	if(pT->m_npListen->status==32602){pT->Close(pT,pT->m_npListen->ident);};
	if(pT->m_npListen->status==0)
	{
	 pT->m_bSrvState = DRV_ST_OPEN;
	 return TRUE;
	}
}

_GLOBAL TcpSend_typ sSend;
_GLOBAL INT iCTcpSrvVal,iCTcpSendCh;
//_GLOBAL INT iLnSSend;
BOOL CTcpServer_SendMessage(This,SMESSAGE *pMsg)
{
    DECLARE_MULTI_OPEN(CTcpServer,CCyclicSystem)
	iCTcpSrvVal++;
	//pT->m_blSState = TRUE;
	//pT->AddCRC(pT,TRUE,pMsg);
	pT->m_npSend->pData   = &pMsg->m_sbyInfo[0];
	pT->m_npSend->datalen = pMsg->m_swLen-9;
	TcpSend(pT->m_npSend);
	memcpy(&sSend,pT->m_npSend,sizeof(TcpSend_typ));
	if(pT->m_npSend->status!=0)
	{
	 if(pT->m_npSend->status==32609)
	 {
		 iCTcpSendCh++;
		 pT->CloseSend(pT);
		 pT->CloseRecc(pT);
		 pT->CloseOpen(pT);
		 pT->Disconnect(pT);
	 }
	 pT->m_blSState = FALSE;
	 return FALSE;
    }
	return TRUE;
}
_GLOBAL INT iPSend;
//_GLOBAL INT iLnPSend;
void CTcpServer_PostSend(This)
{
    DECLARE_MULTI_OPEN(CTcpServer,CCyclicSystem)
	iPSend++;
	TcpSend(pT->m_npSend);
	memcpy(&sSend,pT->m_npSend,sizeof(TcpSend_typ));
  	if(pT->m_npSend->status==0)pT->m_blSState = TRUE;
	if(pT->m_npSend->status==32609){iCTcpSendCh++;pT->CloseSend(pT);pT->CloseRecc(pT);pT->CloseOpen(pT);pT->Disconnect(pT);}
}

//_GLOBAL INT iCTcpCliVal;
_GLOBAL INT iCTcpInData;
//_GLOBAL SMESSAGE sMS;

BOOL CTcpServer_GetMessage(This,SMESSAGE *pMsg)
{
    DECLARE_MULTI_OPEN(CTcpServer,CCyclicSystem)
	pT->m_npRecc->pData = &pMsg->m_sbyInfo[0];
	TcpRecv(&pT->m_npRecc);
	memcpy(&sRecc,&pT->m_npRecc,sizeof(TcpRecv_typ));
	if(pT->m_npRecc->status==0)
	{
	 iCTcpInData++;
	 pMsg->m_swLen  = 9 + pT->m_npRecc->recvlen;
	 pMsg->m_sbyFor = DIR_PHTO101;
	 if (pMsg->m_swLen<300) return TRUE; else return FALSE;
	}
	else
    return FALSE;
}
_GLOBAL INT nReceiveThreadTcp,nSendThreadTcp,nSNDUR;
void CTcpServer_SendThread(This)
{
    DECLARE_MULTI_OPEN(CTcpServer,CCyclicSystem)
	nSendThreadTcp++;
	if(pT->m_bSrvState==DRV_ST_CONN)
    {
	 if(pT->m_blSState==FALSE)
	 	 pT->PostSend(pT);else
	 if(FGET(DEV_TCPBF_BOX_ID,&pT->m_sMsg0))
	 {
	  //Info("\n(__)CTcpR::>TX:%M",&pT->m_sMsg);
	  nSNDUR++;
	  pT->AddCRC(pT,TRUE,&pT->m_sMsg0);
      pT->SendMessage(pT,&pT->m_sMsg0);
	 }
	}
}
_GLOBAL INT nCheckOpenTcp,nCheckSendCheck;
void CTcpServer_ReceiveThread(This)
{
    DECLARE_MULTI_OPEN(CTcpServer,CCyclicSystem)
	nReceiveThreadTcp++;
	if(pT->m_bSrvState==DRV_ST_CONN)
	if(pT->GetMessage(pT,&pT->m_sMsg)==TRUE)
	{
	  nCheckOpenTcp = 0;
	  pT->m_nConnTMR.OnTimer(&pT->m_nConnTMR,100);
	  //Info("\n(__)CTCPM::>RX:%M",&pT->m_sMsg);
	  if(pT->CheckCRC(pT,FALSE,&pT->m_sMsg)==TRUE)
	  {
	   pT->m_sMsg.m_swLen -= 4;
	   pT->m_sMsg.m_sbyFrom       = DIR_PHMDL;
	   pT->m_sMsg.m_sbyFor        = DIR_PHTOMS;
	   pT->m_sMsg.m_sbyIntType    = 0;
	   pT->m_sMsg.m_sbyServerID   = 0;
	   pT->m_sMsg.m_sbyType       = PH_SCMD_REQ;
	   pT->m_sMsg.m_sbyDirection  = 0;
	   pT->m_sMsg.m_sbySensor     = 0;
       FPUT(DEV_MSMDL_BOX_ID,(BYTE*)&pT->m_sMsg);
	  }
	}
}
//_GLOBAL INT iPRecv;
BOOL CTcpServer_PostGet(This)
{
    DECLARE_MULTI_OPEN(CTcpServer,CCyclicSystem)
	return FALSE;
}
//_GLOBAL Tcpclose_typ sClose;
BOOL CTcpServer_Close(This,UDINT uModule)
{
    DECLARE_MULTI_OPEN(CTcpServer,CCyclicSystem)
    BOOL res = TRUE;
	pT->m_bSrvState      = DRV_ST_DISC;
	pT->m_npClose->enable = TRUE;
	pT->m_npClose->ident  = uModule;
	pT->m_npClose->how    = 3;
	TcpClose(pT->m_npClose);
	//pT->Init(pT,pT->m_pArm);
	//memcpy(&sClose,pT->m_npClose,sizeof(Tcpclose_typ));
	if(pT->m_npClose->status==0)return TRUE;
    return FALSE;
}
BOOL CTcpServer_CloseOpen(This)
{
    DECLARE_MULTI_OPEN(CTcpServer,CCyclicSystem)
	BOOL res =pT->Close(pT,pT->m_npListen->ident);
	pT->m_bSrvState = DRV_ST_DISC;
	memset(pT->m_npSend,0,sizeof(TcpSend_typ));
	return res;
}
BOOL CTcpServer_CloseSend(This)
{
    DECLARE_MULTI_OPEN(CTcpServer,CCyclicSystem)
	BOOL res =pT->Close(pT,pT->m_npSend->ident);
	pT->m_bSrvState = DRV_ST_DISC;
	memset(pT->m_npSend,0,sizeof(TcpSend_typ));
	memset(&sSend,0,sizeof(TcpRecv_typ));
	return res;
}
BOOL CTcpServer_CloseRecc(This)
{
    DECLARE_MULTI_OPEN(CTcpServer,CCyclicSystem)
	BOOL res = pT->Close(pT,pT->m_npRecc->ident);
	pT->m_bSrvState = DRV_ST_DISC;
	memset(&pT->m_npRecc,0,sizeof(TcpRecv_typ));
	memset(&sRecc,0,sizeof(TcpRecv_typ));
    return res;
}
BOOL CTcpServer_CheckSend(This)
{
    DECLARE_MULTI_OPEN(CTcpServer,CCyclicSystem)
    return TRUE;
}
void CTcpServer_WordXCHG(This,SMESSAGE *pMsg)
{
	DECLARE_MULTI_OPEN(CTcpServer,CCyclicSystem)
    #ifndef WIN32
	BYTE byTmp,*pW = (BYTE*)pMsg;
	byTmp = pW[0];
	pW[0] = pW[1];
	pW[1] = byTmp;
    #endif
}
BOOL CTcpServer_CheckCRC(This,BOOL blCrc,SMESSAGE *pMsg)
{
	DECLARE_MULTI_OPEN(CTcpServer,CCyclicSystem)
	DWORD dwCrc = 0;
	WORD wLen = pMsg->m_swLen;
	BYTE *pR = (BYTE*)&dwCrc;
	BYTE *pM = (BYTE*)pMsg;
	BYTE *pCRC = &pM[wLen-4];
    #ifndef WIN32
	pR[3] = pCRC[0];
	pR[2] = pCRC[1];
	pR[1] = pCRC[2];
	pR[0] = pCRC[3];
    #else
	memcpy(&dwCrc,pCRC,4);
    #endif
	if(dwCrc==pT->ClcCRC(pT,blCrc,pMsg)) return TRUE;
	return FALSE;
}
DWORD CTcpServer_ClcCRC(This,BOOL blCrc,SMESSAGE *pMsg)
{
    DECLARE_MULTI_OPEN(CTcpServer,CCyclicSystem)
	WORD i;
	WORD wLen;
	DWORD dwCrc = 0;
	//BYTE *pCRC,*pM = (BYTE*)&pMsg;
	BYTE *pCRC,*pM = (BYTE*)&pMsg->m_sbyInfo[0];
	if (blCrc) pMsg->m_swLen += 4;
	//wLen = pMsg->m_swLen-4;
	wLen = pMsg->m_swLen-4-9;
	pCRC = &pM[wLen];
	for(i=0;i<wLen;i++)
	{
	 dwCrc += pM[i];
	 if(i>700)
		 break;
	}
	return dwCrc;
}
void CTcpServer_AddCRC(This,BOOL blCrc,SMESSAGE *pMsg)
{
	DECLARE_MULTI_OPEN(CTcpServer,CCyclicSystem)
	DWORD dwCrc = 0;
	WORD wLen = pMsg->m_swLen;
	BYTE *pR = (BYTE*)&dwCrc;
	BYTE *pM = (BYTE*)pMsg;
	BYTE *pCRC = &pM[wLen];
	dwCrc = pT->ClcCRC(pT,blCrc,pMsg);
    #ifndef WIN32
	pCRC[3] = pR[0];
	pCRC[2] = pR[1];
	pCRC[1] = pR[2];
	pCRC[0] = pR[3];
    #else
	memcpy(pCRC,pR,4);
    #endif
}

BOOL CTcpServer_EventHandler(This,SMESSAGE *pMsg)
{
    DECLARE_MULTI_OPEN(CTcpServer,CCyclicSystem)
	//SHORTMESSAGE m_sMsg;
	switch(pMsg->m_sbyFor)
	{
      case DIR_MSTOTCP:
	       #ifdef DEB_CTcpServer
		   Info("\n(__)CTCPR::>OUTP::%M",pMsg);
		   #endif
		   FPUT(DEV_TCPBF_BOX_ID,pMsg);
	  break;
	  case DIR_TCPTOTCP:
	       if (pMsg->m_sbyType==EV_TMR_SRR_REQ)
		   {

 		    pT->Open(pT);
			pT->m_nConnTMR.OnTimer(&pT->m_nConnTMR,100);
			//if (nCheckOpenTcp%4==0)
			{
             nCheckSendCheck++;
			 pT->m_sMsg0.m_swLen      = 9+3;
			 pT->m_sMsg0.m_sbyInfo[0] = 0x55;
			 pT->m_sMsg0.m_sbyInfo[1] = 0xaa;
			 pT->m_sMsg0.m_sbyInfo[2] = 0x55;
			 pT->m_sMsg0.m_sbyInfo[3] = 3;
			 pT->m_sMsg0.m_sbyInfo[4] = 4;
			 ////SendMessage()
			 FPUT(DEV_TCPBF_BOX_ID,&pT->m_sMsg0);
			}
			nCheckOpenTcp++;
		   }
	  break;
	  default:
	  break;
	}
	return TRUE;
}
void CTcpServer_CyclicProc(This)
{
    DECLARE_MULTI_OPEN(CTcpServer,CCyclicSystem)
    #ifndef WIN32
	pT->SendThread(pT);
	pT->ReceiveThread(pT);
    #else
	pT->SendThread(pT);
    #endif
}
void CTcpServer_SendSMessage(This,BYTE byBox,BYTE byFor,BYTE byType)
{
    DECLARE_MULTI_OPEN(CTcpServer,CCyclicSystem)
	SHORTMESSAGE m_sMsg;
	m_sMsg.m_swLen        = 9;
	m_sMsg.m_sbyFrom      = DIR_PHMDL;
	m_sMsg.m_sbyFor       = byFor;
	m_sMsg.m_sbyIntType   = 0;
	m_sMsg.m_sbyServerID  = 0;
	m_sMsg.m_sbyType      = byType;
	m_sMsg.m_sbyDirection = 0;
	m_sMsg.m_sbySensor    = 0;
	FPUT(byBox,(BYTE*)&m_sMsg);
    #ifdef DEB_CTcpServer
	Info("\n(__)CTCPR::>OUTT::%M",&m_sMsg);
    #endif
}
void CTcpServer_Connect(This)
{
    DECLARE_MULTI_OPEN(CTcpServer,CCyclicSystem)
    SHORTMESSAGE m_sMsg;
	m_sMsg.m_swLen        = 9;
	m_sMsg.m_sbyFrom      = DIR_PHMDL;
	m_sMsg.m_sbyFor       = DIR_PHTO101P;
	m_sMsg.m_sbyIntType   = 0;
	m_sMsg.m_sbyServerID  = 0;
	m_sMsg.m_sbyType      = PH_CONN_IND;
	m_sMsg.m_sbyDirection = 0;
	m_sMsg.m_sbySensor    = 0;
	FPUT(DEV_101MD_BOX_ID,(BYTE*)&m_sMsg);
    #ifdef DEB_CTcpServer
	Info("\n(__)CTCPR::>OUTT::%M",&m_sMsg);
    #endif
}
void CTcpServer_Disconnect(This)
{
    DECLARE_MULTI_OPEN(CTcpServer,CCyclicSystem)
    SHORTMESSAGE m_sMsg;
	m_sMsg.m_swLen        = 9;
	m_sMsg.m_sbyFrom      = DIR_PHMDL;
	m_sMsg.m_sbyFor       = DIR_PHTO101P;
	m_sMsg.m_sbyIntType   = 0;
	m_sMsg.m_sbyServerID  = 0;
	m_sMsg.m_sbyType      = PH_DISC_IND;
	m_sMsg.m_sbyDirection = 0;
	m_sMsg.m_sbySensor    = 0;
	FPUT(DEV_101MD_BOX_ID,(BYTE*)&m_sMsg);
    #ifdef DEB_CTcpServer
	Info("\n(__)CTCPR::>OUTT::%M",&m_sMsg);
    #endif
}
void CTcpServer_CTcpServer(This)
{
    DECLARE_MULTI_OPEN(CTcpServer,CCyclicSystem)
	DECLARE_REGISTRATION(CTcpServer,Init)
	DECLARE_REGISTRATION(CTcpServer,PostSend)
	DECLARE_REGISTRATION(CTcpServer,PostGet)
	DECLARE_REGISTRATION(CTcpServer,SendMessage)
	DECLARE_REGISTRATION(CTcpServer,GetMessage)
	DECLARE_REGISTRATION(CTcpServer,CheckSend)
	DECLARE_REGISTRATION(CTcpServer,Open)
	DECLARE_REGISTRATION(CTcpServer,Listen)
	DECLARE_REGISTRATION(CTcpServer,Close)
	DECLARE_REGISTRATION(CTcpServer,CloseSend)
	DECLARE_REGISTRATION(CTcpServer,CloseRecc)
	DECLARE_REGISTRATION(CTcpServer,WordXCHG)
	DECLARE_REGISTRATION(CTcpServer,AddCRC)
	DECLARE_REGISTRATION(CTcpServer,CheckCRC)
	DECLARE_REGISTRATION(CTcpServer,ClcCRC)
	DECLARE_REGISTRATION(CTcpServer,ReceiveThread)
	DECLARE_REGISTRATION(CTcpServer,SendThread)
	DECLARE_REGISTRATION(CTcpServer,CloseOpen)
	DECLARE_REGISTRATION(CTcpServer,Connect)
	DECLARE_REGISTRATION(CTcpServer,Disconnect)
	DECLARE_REGISTRATION(CTcpServer,SendSMessage)
	DECLARE_VIRTUAL_FUNC(CTcpServer,EventHandler)
	DECLARE_VIRTUAL_FUNC(CTcpServer,CyclicProc)
}
void CTcpServer_DCTcpServer(This)
{
	DECLARE_MULTI_OPEN(CTcpServer,CCyclicSystem)
}
DECLARE_MULTI_CREATE(CTcpServer,CCyclicSystem)
#ifdef WIN32
DWORD WINAPI GetArm(PVOID pVoid)
{
	CTcpServer *pT = (CTcpServer*)pVoid;
	while(1)
	{
	 pT->ReceiveThread(pT);
	 //pT->SendThread(pT);
	 //Sleep(50);
     //printf("\nGetArm");
	}
	return 0;
}
#endif
```
